// TIA Portal project "立体仓库与堆垛系统_V18" (V18)

(* hardware
DEVICE "S7-1200 station_1"  S7-1200 Station
   slot 0: "Rack_0"  S7-1200 Rack  Rack  V1.0
   slot 1: "PLC_1"  CPU 1214C DC/DC/DC  6ES7 214-1AG31-0XB0  V3.0
DEVICE "HMI_1"  TP700 Comfort
   slot 0: "HMI_1"  TP700 Comfort  6AV2 124-0GC01-0AX0  16.0.0.0
   slot 1: "HMI_RT_1"  TP700 Comfort  6AV2 124-0GC01-0AX0  16.0.0.0
   slot 5: "HMI_1.IE_CP_1"  PROFINET Interface  16.0.0.0
      slot 1: "PROFINET Interface_1"  PROFINET Interface
         slot 1: "Port_1"  Port
         slot 2: "Port_2"  Port
   slot 7: "HMI_1.MPI/DP_CP_1"  MPI/DP Interface  16.0.0.0
DEVICE "GSD device_1"  GSD.Device.PN
   slot 0: "机架"  Rack  V1.0
   slot 0: "gl20-pn"  GL20  INOVANCE GL20-PN
      slot 0: "Standard, 1 port"  Standard, 1 port
      slot 1: "Interface"  Interface
         slot 1: "Port 1"  Port 1
         slot 2: "Port 2"  Port 2
   slot 1: " 1600END_1"  1600END
      slot 0: " 1600END"  1600END
   slot 2: " 1600END_2"  1600END
      slot 0: " 1600END"  1600END
   slot 3: " 0800END_1"  0800END
      slot 0: " 0800END"  0800END
   slot 4: " 0016ETN_1"  0016ETN
      slot 0: " 0016ETN"  0016ETN
DEVICE "GSD device_2"  GSD.Device.PN
   slot 0: "机架"  Rack  V1.0
   slot 0: "GL20-pn2"  GL20  INOVANCE GL20-PN
      slot 0: "Standard, 1 port"  Standard, 1 port
      slot 1: "Interface"  Interface
         slot 1: "Port 1"  Port 1
         slot 2: "Port 2"  Port 2
   slot 1: " 1600END_1"  1600END
      slot 0: " 1600END"  1600END
   slot 2: " 0800END_1"  0800END
      slot 0: " 0800END"  0800END
   slot 3: " 0016ETN_1"  0016ETN
      slot 0: " 0016ETN"  0016ETN
*)

// ===== PLC "PLC_1"  CPU 1214C DC/DC/DC =====

VAR_GLOBAL   // PLC tag table "默认变量表"
   "上升按钮" AT %I4.5 : Bool;
   "下降按钮" AT %I4.4 : Bool;
   "自动手动切换按钮" AT %I5.4 : Bool;
   "进货台正转按钮" AT %I4.0 : Bool;
   "进货链运行按钮" AT %I4.1 : Bool;
   "向后按钮" AT %I4.2 : Bool;
   "向前按钮" AT %I4.3 : Bool;
   "右移按钮" AT %I4.6 : Bool;
   "左移按钮" AT %I4.7 : Bool;
   "进货台反转按钮" AT %I5.0 : Bool;
   "出货链运行按钮" AT %I5.1 : Bool;
   "出货台正转按钮" AT %I5.2 : Bool;
   "出货台反转按钮" AT %I5.3 : Bool;
   "Encoder A pulse" AT %I0.0 : Bool;
   "Encoder B pulse" AT %I0.2 : Bool;
   "Shipment in place detection" AT %I2.2 : Bool;
   "enter table limit position" AT %I2.3 : Bool;
   "enter table Zero position" AT %I2.4 : Bool;
   "Incoming goods in place detection" AT %I2.5 : Bool;
   "Left limit of x-axis" AT %I2.6 : Bool;
   "Lower limit of y-axis" AT %I2.7 : Bool;
   "Platform front and back position judgment" AT %I3.0 : Bool;
   "Platform median detection" AT %I3.1 : Bool;
   "Platform behind Limit Position" AT %I3.2 : Bool;
   "Platform Front Limit Position" AT %I3.3 : Bool;
   "Right limit x-axis" AT %I3.4 : Bool;
   "shipping table  Zero position" AT %I3.5 : Bool;
   "shipping table  limit position" AT %I3.6 : Bool;
   "highlimit y-axis" AT %I3.7 : Bool;
   "急停按钮" AT %I5.5 : Bool;
   "16.space in" AT %I6.0 : Bool;   // 16仓库输入
   "15.space in" AT %I6.1 : Bool;   // 15仓库输入
   "14.space in" AT %I6.2 : Bool;   // 14仓库输入
   "13.space in" AT %I6.3 : Bool;   // 13仓库输入
   "4.space in" AT %I6.4 : Bool;   // 4仓库输入
   "3.space in" AT %I6.5 : Bool;   // 3仓库输入
   "2.space in" AT %I6.6 : Bool;   // 2仓库输入
   "1.space in" AT %I6.7 : Bool;   // 1仓库输入
   "Y-axis stepping pulse" AT %Q0.2 : Bool;
   "Y-axis stepping direction" AT %Q0.3 : Bool;
   "High scan" AT %Q3.4 : Bool;
   "Low scan" AT %Q3.2 : Bool;
   "Mid scan" AT %Q3.3 : Bool;
   "进货台逆时针" AT %Q2.3 : Bool;
   "进货台顺时针" AT %Q2.2 : Bool;
   "进货台电机驱动" AT %Q2.4 : Bool;
   "平台向后运行" AT %Q2.1 : Bool;
   "平台向前运行" AT %Q2.0 : Bool;
   "轴向右运行" AT %Q2.6 : Bool;
   "轴向左运行" AT %Q2.5 : Bool;
   "出货台电机驱动" AT %Q3.1 : Bool;
   "出货台顺时针" AT %Q2.7 : Bool;
   "出货台逆时针" AT %Q3.0 : Bool;
   "步进电机硬件限位辅助" AT %Q3.5 : Bool;
   "Enable manual" AT %M0.4 : Bool;
   "Alarm level" AT %MB100 : Byte;
   "Alarm level 1" AT %M101.0 : Bool;
   "Alarm level 2" AT %M101.1 : Bool;
   "Disconnect Automatic" AT %M101.2 : Bool;
   "Emergency stop system" AT %M101.3 : Bool;
   "组态报警" AT %M101.4 : Bool;
   "触摸屏进入自动" AT %M0.1 : Bool;
   "automatic mode" AT %M0.0 : Bool;
   "manual mode" AT %M0.2 : Bool;
   "stoprightnow" AT %M0.3 : Bool;
   "outover" AT %M0.5 : Bool;
   "inover" AT %M0.6 : Bool;
   "outrequests" AT %M0.7 : Bool;
   "inrequests" AT %M1.0 : Bool;
   "inmod" AT %M1.1 : Bool;
   "outmod" AT %M1.2 : Bool;
   "Warehouse vacancies" AT %M1.3 : Bool;
   "space1" AT %M2.0 : Bool;   // 仓口1
   "space2" AT %M2.1 : Bool;
   "space3" AT %M2.2 : Bool;
   "space4" AT %M2.3 : Bool;
   "space5" AT %M2.4 : Bool;
   "space6" AT %M2.5 : Bool;
   "space7" AT %M2.6 : Bool;
   "space8" AT %M2.7 : Bool;
   "space9" AT %M3.0 : Bool;
   "space10" AT %M3.1 : Bool;
   "space11" AT %M3.2 : Bool;
   "space12" AT %M3.3 : Bool;
   "space13" AT %M3.4 : Bool;
   "space14" AT %M3.5 : Bool;
   "space15" AT %M3.6 : Bool;
   "space16" AT %M3.7 : Bool;
   "space17" AT %M4.0 : Bool;
   "space18" AT %M4.1 : Bool;
   "space19" AT %M4.2 : Bool;
   "space20" AT %M4.3 : Bool;
   "shelf1.NO1" AT %MB2 : USInt;
   "shelf1.NO2" AT %MB3 : USInt;
   "shelf2" AT %MB4 : USInt;
   "移动至货仓8" AT %M10.0 : Bool;
   "移动至货仓7" AT %M10.1 : Bool;
   "移动至货仓6" AT %M10.2 : Bool;
   "移动至货仓5" AT %M10.3 : Bool;
   "移动至货仓4" AT %M10.4 : Bool;
   "移动至货仓3" AT %M10.5 : Bool;
   "移动至货仓2" AT %M10.6 : Bool;
   "移动至货仓1" AT %M10.7 : Bool;
   "移动至货仓16" AT %M11.0 : Bool;
   "移动至货仓15" AT %M11.1 : Bool;
   "移动至货仓14" AT %M11.2 : Bool;
   "移动至货仓13" AT %M11.3 : Bool;
   "移动至货仓12" AT %M11.4 : Bool;
   "移动至货仓11" AT %M11.5 : Bool;
   "移动至货仓10" AT %M11.6 : Bool;
   "移动至货仓9" AT %M11.7 : Bool;
   "移动至货仓17" AT %M12.0 : Bool;
   "移动至货仓18" AT %M12.1 : Bool;
   "移动至货仓19" AT %M12.2 : Bool;
   "移动至货仓20" AT %M12.3 : Bool;
   "backhome" AT %M200.0 : Bool;
   "higher limit of y-axis.sav" AT %M320.2 : Bool;
   "manual_up" AT %M200.3 : Bool;
   "Manual_descent" AT %M200.4 : Bool;
   "Setting Y displacement" AT %MD210 : Real;
   "frontbackO" AT %M13.0 : Bool;
   "behindbackO" AT %M13.1 : Bool;
   "frontlimitgo" AT %M13.2 : Bool;
   "behindlimitgo" AT %M13.3 : Bool;
   "front and back pos judge.sav" AT %M13.4 : Bool;
   "停止回原点前半边" AT %M13.6 : Bool;   // +
   "停止回原点后半轴" AT %M13.7 : Bool;
   "平台前后位判断存(1)" AT %M14.0 : Bool;
   "Pulse A-encoder value" AT %ID1000 : UDInt;
   "Setting X displacement" AT %MD220 : UDInt;
   "insteps.sav" AT %MB5 : USInt;
   "instep1" AT %M15.0 : Bool;
   "instep2" AT %M15.1 : Bool;
   "instep3" AT %M15.2 : Bool;
   "instep4" AT %M15.3 : Bool;
   "instep5" AT %M15.4 : Bool;
   "自动回原点上升" AT %M200.5 : Bool;
   "绝对位移" AT %M200.6 : Bool;
   "回相对原点O" AT %M200.7 : Bool;
   "向O上升" AT %M6.0 : Bool;
   "远O下降" AT %M6.1 : Bool;
   "确认复位" AT %M6.2 : Bool;
   "Tag_1" AT %M17.0 : Bool;
   "调试专用" AT %M9.0 : Bool;
   "Z轴电机初始态完成" AT %M8.1 : Bool;
   "限制使用现场手自动" AT %M1.4 : Bool;
   "AUTO/manual" AT %M1.5 : Bool;
   "in_Pick Pos Completion" AT %M8.0 : Bool;
   "X auto left" AT %M7.0 : Bool;
   "X auto right" AT %M7.1 : Bool;
   "X-axis motion end" AT %M7.2 : Bool;
   "Y-axis motion end" AT %M7.3 : Bool;
   "X-axis right motion lock" AT %M7.4 : Bool;
   "X-axis left motion lock" AT %M7.5 : Bool;
   "instep6" AT %M15.5 : Bool;
   "instep7" AT %M15.6 : Bool;
   "AUTObehindlimitgo" AT %M7.6 : Bool;
   "AUTObehindbackO" AT %M7.7 : Bool;
   "AUTOfrontlimitgo" AT %M14.1 : Bool;
   "AUTOfrontbackO" AT %M14.2 : Bool;
   "停止轴" AT %M8.2 : Bool;
   "instep8" AT %M15.7 : Bool;
   "instep9" AT %M16.0 : Bool;
   "instep10" AT %M16.1 : Bool;
   "步进电机绝对位移ERROR-ID" AT %MD1000 : DWord;
   "Y_coordinate" AT %MD230 : Real;
   "X_coordinate" AT %MD240 : UDInt;
   "Tscan_over" AT %M17.1 : Bool;
   "Tscan_ET" AT %MD1004 : Time;
   "LV.highset" AT %M17.2 : Bool;
   "LV.midset" AT %M17.3 : Bool;
   "LV.lowset" AT %M17.4 : Bool;
   "instep11" AT %M16.2 : Bool;
   "endLOCAT.X" AT %MD250 : UDInt;
   "endLOCAT.Y" AT %MD260 : Real;
   "instep12" AT %M16.3 : Bool;
   "instep13" AT %M16.4 : Bool;
   "instep14" AT %M16.5 : Bool;
   "instep15" AT %M16.6 : Bool;
   "LOWTIME" AT %MD270 : Time;
   "MIDTIME" AT %MD274 : Time;
   "HIGHTIME" AT %MD278 : Time;
   "mov_to1" AT %M110.0 : Bool;   // 人机交互-组态
   "mov_to2" AT %M110.1 : Bool;
   "mov_to3" AT %M110.2 : Bool;
   "mov_to4" AT %M110.3 : Bool;
   "mov_to5" AT %M110.4 : Bool;
   "mov_to6" AT %M110.5 : Bool;
   "mov_to7" AT %M110.6 : Bool;
   "mov_to8" AT %M110.7 : Bool;
   "mov_to9" AT %M111.0 : Bool;
   "mov_to10" AT %M111.1 : Bool;
   "mov_to11" AT %M111.2 : Bool;
   "mov_to12" AT %M111.3 : Bool;
   "mov_to13" AT %M111.4 : Bool;
   "mov_to14" AT %M111.5 : Bool;
   "mov_to15" AT %M111.6 : Bool;
   "mov_to16" AT %M111.7 : Bool;
   "mov_to17" AT %M112.0 : Bool;
   "mov_to18" AT %M112.1 : Bool;
   "mov_to19" AT %M112.2 : Bool;
   "mov_to20" AT %M112.3 : Bool;
   "outgoodsexist" AT %M17.5 : Bool;
   "outsteps.sav" AT %MB18 : USInt;
   "outstep1" AT %M19.0 : Bool;
   "outstep2" AT %M19.1 : Bool;
   "outstep3" AT %M19.2 : Bool;
   "outstep4" AT %M19.3 : Bool;
   "outstep5" AT %M19.4 : Bool;
   "outstep6" AT %M19.5 : Bool;
   "outstep7" AT %M19.6 : Bool;
   "outstep8" AT %M19.7 : Bool;
   "outstep9" AT %M20.0 : Bool;
   "outstep10" AT %M20.1 : Bool;
   "outstep11" AT %M20.2 : Bool;
   "outstep12" AT %M20.3 : Bool;
   "outstep13" AT %M20.4 : Bool;
   "outstep14" AT %M20.5 : Bool;
   "outstep15" AT %M20.6 : Bool;
   "out_Pick Pos Completion" AT %M17.6 : Bool;
   "opt_interrupt" AT %M17.7 : Bool;
   "outstep16" AT %M20.7 : Bool;
   "inset_running" AT %M21.0 : Bool;
   "outget_running" AT %M21.1 : Bool;
   "WillLOCAT.X" AT %MD282 : UDInt;
   "WillLOCAT.Y" AT %MD286 : Real;
   "error_goodslose(out.mod)" AT %M21.2 : Bool;
   "OUTlosttime" AT %MD1008 : Time;
   "error_spacewrong(In.mod)" AT %M21.3 : Bool;
   "warn_NOspace(In.mod)" AT %M21.4 : Bool;
   "coverchoicehmi" AT %M21.5 : Bool;
   "INlosttime" AT %MD1012 : Time;
   "error_goodslose(IN.mod)" AT %M21.6 : Bool;
   "error_spacewrong(out.mod)" AT %M21.7 : Bool;
   "进货台正转HMI" AT %M30.0 : Bool;
   "进货台反转HMI" AT %M30.1 : Bool;
   "出货台正转HMI" AT %M30.2 : Bool;
   "出货台反转HMI" AT %M30.3 : Bool;
   "进货链运行HMI" AT %M30.4 : Bool;
   "出货链运行HMI" AT %M30.5 : Bool;
   "左移HMI" AT %M30.6 : Bool;
   "右移HMI" AT %M30.7 : Bool;
   "上升HMI" AT %M31.0 : Bool;
   "下降HMI" AT %M31.1 : Bool;
   "向前HMI" AT %M31.2 : Bool;
   "向后HMI" AT %M31.3 : Bool;
   "System_Byte" AT %MB500 : Byte;
   "启动标志点" AT %M400.0 : Bool;
   "循环标志位" AT %M400.1 : Bool;
   "停止" AT %M400.2 : Bool;
   "复位完成" AT %M400.5 : Bool;
   "Tag_2" AT %M400.4 : Bool;
   "Tag_3" AT %M400.6 : Bool;
   "System_Byte(1)" AT %MB1 : Byte;
   "FirstScan" AT %M500.0 : Bool;
   "DiagStatusUpdate" AT %M500.1 : Bool;
   "AlwaysTRUE" AT %M500.2 : Bool;
   "AlwaysFALSE" AT %M500.3 : Bool;
END_VAR

VAR_GLOBAL   // PLC tag table "gl20-np2输出"
   "进" AT %Q4.0 : Bool;
   "推" AT %Q4.1 : Bool;
   "变频器（黄）" AT %Q4.2 : Bool;
   "链运行" AT %Q4.3 : Bool;
   "码垛升" AT %Q4.4 : Bool;
   "挡板挡" AT %Q4.5 : Bool;
   "平台升" AT %Q4.6 : Bool;
   "放" AT %Q4.7 : Bool;
   "退" AT %Q5.0 : Bool;
   "回" AT %Q5.1 : Bool;
   "变频器（橙）" AT %Q5.2 : Bool;
   "带运行" AT %Q5.3 : Bool;
   "码垛降" AT %Q5.4 : Bool;
   "挡板回" AT %Q5.5 : Bool;
   "平台降" AT %Q5.6 : Bool;
   "货转向" AT %Q5.7 : Bool;
END_VAR

VAR_GLOBAL   // PLC tag table "gl20-np2输入"
   "(n)" AT %I7.0 : Bool;
   "码垛升到位传感器(h)" AT %I7.1 : Bool;
   "码垛到位传感器(b)" AT %I7.2 : Bool;
   "推中到位传感器(d)" AT %I7.3 : Bool;
   "推到位传感器(j)" AT %I7.4 : Bool;
   "码垛下降到位传感器(i)" AT %I7.5 : Bool;
   "平台检测光电传感器(L)" AT %I7.6 : Bool;
   "平台上到位传感器(0)" AT %I7.7 : Bool;
   "挡板挡到位(m)" AT %I8.0 : Bool;
   "码垛输入传感器(a)" AT %I8.1 : Bool;
   "回到位传感器(c)" AT %I8.2 : Bool;
   "推到位传感器(e)" AT %I8.3 : Bool;
   "退到位传感器(f)" AT %I8.4 : Bool;
   "码垛高度匹配传感器(g)" AT %I8.5 : Bool;
   "平台到位传感器(k)" AT %I8.6 : Bool;
   "平台下到位传感器(p)" AT %I8.7 : Bool;
   "手动自动" AT %I9.0 : Bool;
END_VAR

DATA_BLOCK "Locat"   // DB11
{ S7_Optimized_Access := 'TRUE' }
VERSION : 0.1
   VAR RETAIN
      "shelf  X axis" : Array[0..19] of UDInt;
      "shelf  Y axis" : Array[0..19] of Real;
   END_VAR
BEGIN
   "shelf  X axis"[0] := 1362;
   "shelf  X axis"[1] := 1362;
   "shelf  X axis"[2] := 1061;
   "shelf  X axis"[3] := 1061;
   "shelf  X axis"[4] := 929;
   "shelf  X axis"[5] := 929;
   "shelf  X axis"[6] := 929;
   "shelf  X axis"[7] := 764;
   "shelf  X axis"[8] := 764;
   "shelf  X axis"[9] := 633;
   "shelf  X axis"[10] := 633;
   "shelf  X axis"[11] := 633;
   "shelf  X axis"[12] := 466;
   "shelf  X axis"[13] := 466;
   "shelf  X axis"[14] := 334;
   "shelf  X axis"[15] := 334;
   "shelf  X axis"[16] := 334;
   "shelf  X axis"[17] := 34;
   "shelf  X axis"[18] := 34;
   "shelf  X axis"[19] := 34;
   "shelf  Y axis"[0] := -263.0;
   "shelf  Y axis"[1] := -130.0;
   "shelf  Y axis"[6] := 2.5;
   "shelf  Y axis"[5] := -130.0;
   "shelf  Y axis"[4] := -263.0;
   "shelf  Y axis"[3] := -130.0;
   "shelf  Y axis"[2] := -263.0;
   "shelf  Y axis"[7] := -263.0;
   "shelf  Y axis"[8] := -130.0;
   "shelf  Y axis"[9] := -263.0;
   "shelf  Y axis"[10] := -130.0;
   "shelf  Y axis"[11] := 2.5;
   "shelf  Y axis"[12] := -263.0;
   "shelf  Y axis"[13] := -130.0;
   "shelf  Y axis"[14] := -263.0;
   "shelf  Y axis"[15] := -130.0;
   "shelf  Y axis"[16] := 2.5;
   "shelf  Y axis"[17] := -263.0;
   "shelf  Y axis"[18] := -130.0;
   "shelf  Y axis"[19] := 2.5;
END_DATA_BLOCK

DATA_BLOCK "mov choice"   // DB12
{ S7_Optimized_Access := 'TRUE' }
VERSION : 0.1
   VAR RETAIN
      NO : Array[0..19] of Bool;
   END_VAR
   VAR
      i : USInt;
      WZ : USInt;
   END_VAR
BEGIN
END_DATA_BLOCK

// folder: System blocks/Program resources

DATA_BLOCK "复位协助z轴"   // DB7
{ S7_Optimized_Access := 'TRUE' }
AUTHOR : Simatic
FAMILY : IEC
NAME : IEC_TMR
VERSION : 1.0
// stored: InstanceOfName IEC_TIMER
"IEC_TIMER"
BEGIN
END_DATA_BLOCK

DATA_BLOCK "脉冲定时底"   // DB8
{ S7_Optimized_Access := 'TRUE' }
AUTHOR : Simatic
FAMILY : IEC
NAME : IEC_TMR
VERSION : 1.0
// stored: InstanceOfName IEC_TIMER
"IEC_TIMER"
BEGIN
END_DATA_BLOCK

DATA_BLOCK "脉冲定时中"   // DB9
{ S7_Optimized_Access := 'TRUE' }
AUTHOR : Simatic
FAMILY : IEC
NAME : IEC_TMR
VERSION : 1.0
// stored: InstanceOfName IEC_TIMER
"IEC_TIMER"
BEGIN
END_DATA_BLOCK

DATA_BLOCK "脉冲定时高"   // DB10
{ S7_Optimized_Access := 'TRUE' }
AUTHOR : Simatic
FAMILY : IEC
NAME : IEC_TMR
VERSION : 1.0
// stored: InstanceOfName IEC_TIMER
"IEC_TIMER"
BEGIN
END_DATA_BLOCK

DATA_BLOCK "time_scan_houseware"   // DB13
{ S7_Optimized_Access := 'TRUE' }
AUTHOR : Simatic
FAMILY : IEC
NAME : IEC_TMR
VERSION : 1.0
// stored: InstanceOfName IEC_TIMER
"IEC_TIMER"
BEGIN
END_DATA_BLOCK

DATA_BLOCK "NOgoodsTON"   // DB15
{ S7_Optimized_Access := 'TRUE' }
AUTHOR : Simatic
FAMILY : IEC
NAME : IEC_TMR
VERSION : 1.0
// stored: InstanceOfName IEC_TIMER
"IEC_TIMER"
BEGIN
END_DATA_BLOCK

// folder: 堆垛系统

DATA_BLOCK "数据块"   // DB16
{ S7_Optimized_Access := 'TRUE' }
VERSION : 0.1
   VAR
      标志位 : Array[1..30] of Bool;
      沿 : Array[1..9] of Bool;
      定时器 : Array[1..6] of IEC_TIMER;
      码垛数量 : Int;
      当前时间 : Time;
      限制 : Bool;
      码垛总数量 : Int;
      余数 : Int;
   END_VAR
BEGIN
END_DATA_BLOCK

DATA_BLOCK "输出数据块"   // DB17
{ S7_Optimized_Access := 'FALSE' }
VERSION : 0.1
   VAR
      带运行 : Bool;
      推 : Bool;
      回1 : Bool;
      回2 : Bool;
      平台降 : Bool;
      平台升1 : Bool;
      平台升2 : Bool;
      放 : Bool;
      链运行 : Bool;
      链运行2 : Bool;
      码垛降 : Bool;
      码垛升1 : Bool;
      码垛升2 : Bool;
      码垛进 : Bool;
      码垛退1 : Bool;
      码垛退2 : Bool;
      挡板挡 : Bool;
      挡板回1 : Bool;
      挡板回2 : Bool;
   END_VAR
BEGIN
END_DATA_BLOCK

// folder: (top level)

DATA_BLOCK "轴_1"   // DB1, Motion_DB
{ S7_Optimized_Access := 'TRUE' }
AUTHOR : SIMATIC
FAMILY : BasicMC
NAME : TO_PTO
VERSION : 3.0
// stored: InstanceOfName TO_Axis_PTO
"TO_Axis_PTO"
BEGIN
   // Axis.OnlinePtoIndexCU = 1
   // Axis.DirectionHwcnAddressCU = Q0.3
   // Axis.PulseHwcnAddressCU = Q0.2
   // Pulse.MinDeltaDeltaFrequencyCU = 0.004
   // Pulse.MaxDeltaDeltaFrequencyCU = 1.0E+10
   // Pulse.MinDeltaFrequencyCU = 0.005
   // Pulse.MaxDeltaFrequencyCU = 9.5E+9
   // Pulse.MinFrequencyCU = 1.0
   // Pulse.MaxFrequencyCU = 100000.0
   // Pulse.OutputSourceCU = 16#0000_0000
   // Axis.SelectPTO = 1
END_DATA_BLOCK

FUNCTION "Auto Out_ware Main Program" : Void   // FC1, SCL
{ S7_Optimized_Access := 'TRUE' }
VERSION : 0.1
BEGIN
   "Shelf Path Selection Subroutine"();//必须进入出库模式才可以访问本页面
   // "opt_interrupt"=1时进入选择，面板变量会,仅在完成正在执行的出库工作或首次使用出库模式后可激活，更新预定的出库序列
   // 不要同时按"movtoxxxx"和"opt_interrupt:=0".此操作不规范，系统会对此进行紧急停止处理。
   IF "outrequests" = 1 AND "outover" = 1 AND "outsteps.sav" = 0 AND "outgoodsexist"AND "opt_interrupt"=0 THEN
       "outsteps.sav" := 1;
       "outover" := 0;
       "coverchoicehmi" := 0;// 关闭选择面板
   END_IF;
   IF "opt_interrupt"=1 AND "outover" = 1 THEN
       "coverchoicehmi" := 1; // 组态里打开选择面板，才可以选择或取消接下来的取货位置
       ;
   END_IF;


   CASE "outsteps.sav" OF
           //取货步
       1:"outstep1" := 1;
           "out_Pick Pos Completion" := "X-axis motion end" AND "Y-axis motion end";
       2:"outstep2" := 1;
       3:"outstep3" := 1;
       4:"outstep4" := 1;
       5:"outstep5" := 1;
       6:"outstep6" := 1;
       7:"outstep7" := 1;
       8:"outstep8" := 1;
       9:"outstep9" := 1;
       10:"outstep10" := 1;
           "out_Pick Pos Completion" := "X-axis motion end" AND "Y-axis motion end";
       11:"outstep11" := 1;
       12:"outstep12" := 1;
       13:"outstep13" := 1;
       14:"outstep14" := 1;
       15:
           "outstep15" := 1;
       16:
           "outstep16" := 1;
       17:
           "outsteps.sav" := 0; // 步序复位
           "outover" := 1;
           IF "outgoodsexist"=0 THEN
               "mov_to13" := 0;
               "mov_to17" := 0;
               "mov_to14" := 0;
               "mov_to18" := 0;
               "mov_to1" := 0;
               "mov_to5" := 0;
               "mov_to9" := 0;
               "mov_to15" := 0;
               "mov_to19" := 0;
               "mov_to2" := 0;
               "mov_to6" := 0;
               "mov_to10" := 0;
               "mov_to16" := 0;
               "mov_to20" := 0;
               "mov_to3" := 0;
               "mov_to7" := 0;
               "mov_to11" := 0;
               "mov_to4" := 0;
               "mov_to8" := 0;
               "mov_to12" := 0;
               // Statement section IF
               ;
           END_IF;
       ELSE
           "outsteps.sav" := 0; // 步序复位
           "outover" := 1;

   END_CASE;

   //出库步序1取货开始
   IF "outstep1" AND ("out_Pick Pos Completion" = 0) THEN
       "Z-axis motor subroutine"();
       IF  "outget_running"=0 OR ("WillLOCAT.X" = "X_coordinate"AND "WillLOCAT.Y" = "Y_coordinate") THEN
           IF "endLOCAT.X" = "X_coordinate" THEN
               // 不需要左右移动直接取
               "Setting Y displacement" := ("Y_coordinate" - 15.0);
               "Y-axis stepper motor subroutine"();
               "X-axis motion end" := 1;
               "WillLOCAT.X" := "X_coordinate";
               "WillLOCAT.Y" := "Y_coordinate";
               "outget_running" := 1;
           ELSE
               //mov后取        
               "Setting X displacement" := "X_coordinate";
               "Setting Y displacement" := ("Y_coordinate" - 15.0);
               "X-axis motor encoder group subroutine"();
               "Y-axis stepper motor subroutine"();
               "WillLOCAT.X" := "X_coordinate";
               "WillLOCAT.Y" := "Y_coordinate";
               "outget_running" := 1;
           END_IF;
       ELSE
           "stoprightnow" := 1;
           "error_spacewrong(out.mod)" := 1;

       END_IF;



   ELSIF "outstep1" AND ("out_Pick Pos Completion" = 1) THEN
       "outstep1" := 0;
       "outsteps.sav" := "outsteps.sav" + 1;
       "Setting Y displacement" := -120;
       "Y-axis stepper motor subroutine"();
       "X-axis motion end" := 0;
       "X-axis left motion lock" := 0;
       "X-axis right motion lock" := 0;
       "Setting X displacement" := 0;
       "endLOCAT.X" :="X_coordinate";
       "endLOCAT.Y" := "Y_coordinate";
       "outget_running" := 0;
   END_IF;
   //出库步序2选择货架
   IF "outstep2" THEN
       IF    "WillLOCAT.X" = "X_coordinate"AND "WillLOCAT.Y" = "Y_coordinate"  THEN
           IF "X_coordinate" = 929 OR "X_coordinate" = 633 OR "X_coordinate" = 334 OR "X_coordinate" = 34 THEN
               "outstep2" := 0;
               "outsteps.sav" := "outsteps.sav" + 4;
           ELSIF "X_coordinate" = 1362 OR "X_coordinate" = 1061 OR "X_coordinate" = 764 OR "X_coordinate" = 466 THEN
               "outstep2" := 0;
               "outsteps.sav" := "outsteps.sav" + 1;
               ;
           END_IF;  // Statement section IF
       ELSE
           "stoprightnow" := 1;
           "error_spacewrong(out.mod)" := 1;
       END_IF;



   END_IF;
       //取货架2
       //出库步序3
       IF "outstep3" AND ("Platform Front Limit Position" = 0) THEN
           "AUTOfrontlimitgo" := 1;
           "Z-axis motor subroutine"();
       ELSIF "outstep3" AND ("Platform Front Limit Position" = 1) THEN
           "AUTOfrontlimitgo" := 0;
           "outstep3" := 0;
           "outsteps.sav" := "outsteps.sav" + 1;
       END_IF;
       //出库步序4
       IF "outstep4" AND ("Y-axis motion end" = 0) THEN
           "Z-axis motor subroutine"();
               "Setting Y displacement" := "Y_coordinate";
               "Y-axis stepper motor subroutine"();
       ELSIF "outstep4" AND ("Y-axis motion end" = 1) THEN
           "outstep4" := 0;
           "outsteps.sav" := "outsteps.sav" + 1;
           "Setting Y displacement" := -120;
           "Y-axis stepper motor subroutine"();
       END_IF;
       //出库步序5
       IF "outstep5" AND ("Platform Front Limit Position" = 1 OR "frontbackO" = 1) THEN
           "AUTOfrontbackO" := 1;
           "Z-axis motor subroutine"();
       ELSIF "outstep5" AND ("Platform Front Limit Position" = 0 AND "frontbackO" = 0) THEN
           "AUTOfrontbackO" := 0;
           "outstep5" := 0;
           "outsteps.sav" := "outsteps.sav" + 4;
       END_IF;
       //取货架1
       //出库步序6
       IF "outstep6" AND ("Platform behind Limit Position" = 0) THEN
           "AUTObehindlimitgo" := 1;
           "Z-axis motor subroutine"();
       ELSIF "outstep6" AND ("Platform behind Limit Position" = 1) THEN
           "AUTObehindlimitgo" := 0;
           "outstep6" := 0;
           "outsteps.sav" := "outsteps.sav" + 1;
       END_IF;
       //出库步序7
       IF "outstep7" AND ("Y-axis motion end" = 0) THEN
           "Z-axis motor subroutine"();
               "Setting Y displacement" := "Y_coordinate";
               "Y-axis stepper motor subroutine"();
       ELSIF "outstep7" AND ("Y-axis motion end" = 1) THEN
           "outstep7" := 0;
           "outsteps.sav" := "outsteps.sav" + 1;
           "Setting Y displacement" := -120;
           "Y-axis stepper motor subroutine"();
       END_IF;
       //出库步序8
       IF "outstep8" AND ("Platform behind Limit Position" = 1 OR "behindbackO" = 1) THEN
           "AUTObehindbackO" := 1;
           "Z-axis motor subroutine"();
       ELSIF "outstep8" AND ("Platform behind Limit Position" = 0 AND "behindbackO" = 0) THEN
           "AUTObehindbackO" := 0;
           "outstep8" := 0;
           "outsteps.sav" := "outsteps.sav" + 1;
       END_IF;
       //出库步序9
       IF "outstep9" AND ("shipping table  Zero position" = 0) THEN
           "出货台逆时针" := 1 AND ("stoprightnow" = 0);
       ELSIF "outstep9" AND ("shipping table  Zero position" = 1) THEN
           "出货台逆时针" := 0;
           "outstep9" := 0;
           "outsteps.sav" := "outsteps.sav" + 1;
       END_IF;
       //出库步序10
       IF "outstep10" AND ("out_Pick Pos Completion" = 0) THEN
           "Z-axis motor subroutine"();
           IF "endLOCAT.X" <= 40 AND "endLOCAT.Y" = 2.5 THEN
               "Setting Y displacement" := -260;
               "Y-axis stepper motor subroutine"();
               "X-axis motion end" := 1;
           ELSIF "endLOCAT.X" <= 40 AND "endLOCAT.Y" = -130.0 THEN
               "Setting Y displacement" := -260;
               "Y-axis stepper motor subroutine"();
               "X-axis motion end" := 1;
           ELSIF "endLOCAT.X" <= 40 AND "endLOCAT.Y" = -263.0 THEN
               "Setting Y displacement" := -263;
               "Y-axis stepper motor subroutine"();
               "X-axis motion end" := 1;
           ELSE
               "Setting X displacement" := 35;
               "Setting Y displacement" := -260;
               "X-axis motor encoder group subroutine"();
               "Y-axis stepper motor subroutine"();

           END_IF;
       ELSIF "outstep10" AND ("out_Pick Pos Completion" = 1) THEN
           "outstep10" := 0;
           "outsteps.sav" := "outsteps.sav" + 1;
           "Setting Y displacement" := -120;
           "Y-axis stepper motor subroutine"();
           "X-axis motion end" := 0;
           "X-axis left motion lock" := 0;
           "X-axis right motion lock" := 0;
           "Setting X displacement" := 0;
       END_IF;
       //出库步序11
       IF "outstep11" AND ("Platform Front Limit Position" = 0) THEN
           "AUTOfrontlimitgo" := 1;
           "Z-axis motor subroutine"();
       ELSIF "outstep11" AND ("Platform Front Limit Position" = 1) THEN
           "AUTOfrontlimitgo" := 0;
           "outstep11" := 0;
           "outsteps.sav" := "outsteps.sav" + 1;
       END_IF;
       //出库步序12
       IF "outstep12" AND ("Y-axis motion end" = 0) THEN
           "Z-axis motor subroutine"();
           "Setting Y displacement" := -278;
           "Y-axis stepper motor subroutine"();
       ELSIF "outstep12" AND ("Y-axis motion end" = 1) THEN
           "outstep12" := 0;
           "outsteps.sav" := "outsteps.sav" + 1;
           "Setting Y displacement" := -120;
           "Y-axis stepper motor subroutine"();
       END_IF;
       //出库步序13
       IF "outstep13" AND ("Platform Front Limit Position" = 1 OR "frontbackO" = 1) THEN
           "AUTOfrontbackO" := 1;
           "Z-axis motor subroutine"();
       ELSIF "outstep13" AND ("Platform Front Limit Position" = 0 AND "frontbackO" = 0) THEN
           "AUTOfrontbackO" := 0;
           "outstep13" := 0;
           "outsteps.sav" := "outsteps.sav" + 1;
       END_IF;
       //出库步序14
       IF "outstep14" AND ("Y-axis motion end" = 0) THEN
           "Z-axis motor subroutine"();
           "Setting Y displacement" := -145;
           "Y-axis stepper motor subroutine"();
       ELSIF "outstep14" AND ("Y-axis motion end") THEN
           "outstep14" := 0;
           "outsteps.sav" := "outsteps.sav" + 1;
           "Setting Y displacement" := -120;
           "Y-axis stepper motor subroutine"();
           "endLOCAT.X" := 34;
           "endLOCAT.Y" := -145;
           "WillLOCAT.X" := 0;
           "WillLOCAT.Y" :=0;
       END_IF;
       //出库步序15
       IF "outstep15" AND ("shipping table  limit position" = 0) THEN
           "出货台顺时针" := 1 AND ("stoprightnow" = 0);
       ELSIF "outstep15" AND ("shipping table  limit position" = 1) THEN
           "出货台顺时针" := 0;
           "outstep15" := 0;
           "outsteps.sav" := "outsteps.sav" + 1;
       END_IF;
       //出库步序16
       "NOgoodsTON".TON(IN := ("outstep16" AND NOT "Shipment in place detection"),
                        PT := T#30s,
                        Q => "error_goodslose(out.mod)",
                        ET => "OUTlosttime");
       IF "outstep16" AND ("Shipment in place detection" = 0) THEN
           "出货台电机驱动" := 1 AND ("stoprightnow" = 0);
           "stoprightnow" := "error_goodslose(out.mod)";
       ELSIF "outstep16" AND ("Shipment in place detection" = 1) THEN
           "出货台电机驱动" := 0;
           "outstep16" := 0;
           "outsteps.sav" := "outsteps.sav" + 1;
       END_IF;
END_FUNCTION

FUNCTION "manual control" : Void   // FC2, LAD
{ S7_Optimized_Access := 'TRUE' }
VERSION : 0.1
BEGIN

REGION Network 1 (SCL)
   //手动切换为自动后必须立即进行复位，禁止不复位而立即请求
   IF "自动手动切换按钮" = 0 THEN
       "outmod" := 0;
       "inmod" := 0;
       "inrequests" := 0;
       "outrequests" := 0;
   END_IF;
END_REGION

REGION Network 2
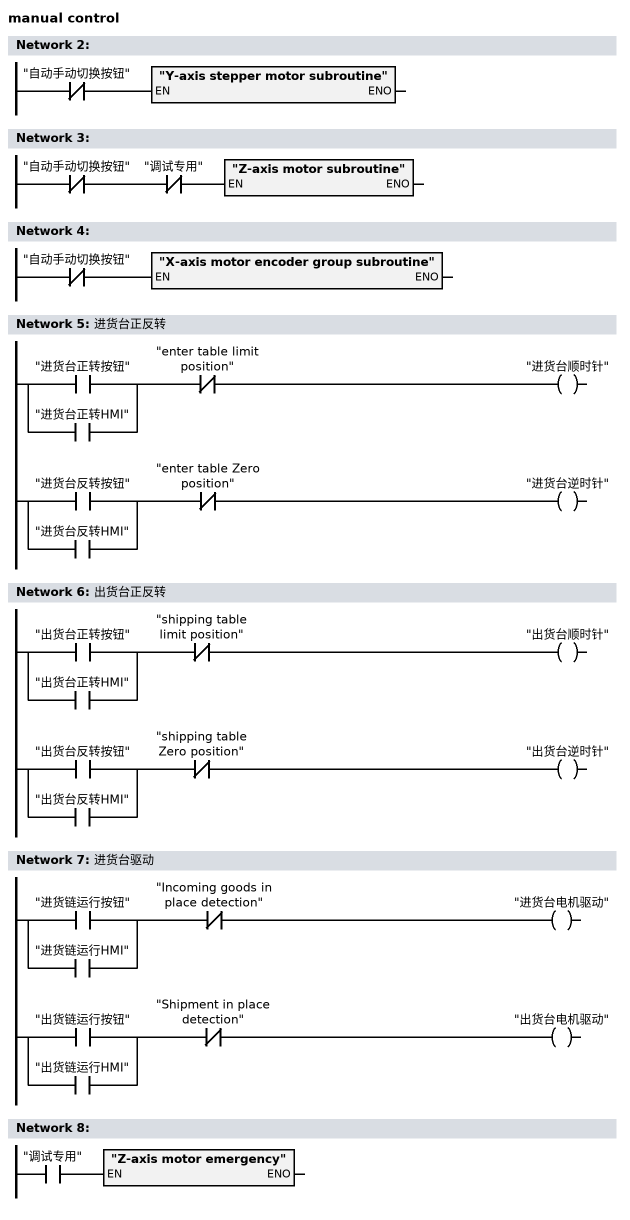
   RUNG wire#powerrail
      I_Contact( "自动手动切换按钮" )
      "Y-axis stepper motor subroutine"()
   END_RUNG
   // the same network as SCL:
   IF NOT "自动手动切换按钮" THEN "Y-axis stepper motor subroutine"(); END_IF;
END_REGION

REGION Network 3
   RUNG wire#powerrail
      I_Contact( "自动手动切换按钮" )
      I_Contact( "调试专用" )
      "Z-axis motor subroutine"()
   END_RUNG
   // the same network as SCL:
   IF NOT "自动手动切换按钮" AND NOT "调试专用" THEN "Z-axis motor subroutine"(); END_IF;
END_REGION

REGION Network 4
   RUNG wire#powerrail
      I_Contact( "自动手动切换按钮" )
      "X-axis motor encoder group subroutine"()
   END_RUNG
   // the same network as SCL:
   IF NOT "自动手动切换按钮" THEN "X-axis motor encoder group subroutine"(); END_IF;
END_REGION

REGION Network 5: 进货台正反转
   RUNG wire#powerrail
      Contact( "进货台正转按钮" )
      wire#w1
      I_Contact( "enter table limit position" )
      Coil( "进货台顺时针" )
   END_RUNG
   RUNG wire#powerrail
      Contact( "进货台正转HMI" )
   END_RUNG wire#w1
   RUNG wire#powerrail
      Contact( "进货台反转按钮" )
      wire#w2
      I_Contact( "enter table Zero position" )
      Coil( "进货台逆时针" )
   END_RUNG
   RUNG wire#powerrail
      Contact( "进货台反转HMI" )
   END_RUNG wire#w2
   // the same network as SCL:
   "进货台顺时针" := ("进货台正转按钮" OR "进货台正转HMI") AND NOT "enter table limit position";
   "进货台逆时针" := ("进货台反转按钮" OR "进货台反转HMI") AND NOT "enter table Zero position";
END_REGION

REGION Network 6: 出货台正反转
   RUNG wire#powerrail
      Contact( "出货台正转按钮" )
      wire#w1
      I_Contact( "shipping table  limit position" )
      Coil( "出货台顺时针" )
   END_RUNG
   RUNG wire#powerrail
      Contact( "出货台正转HMI" )
   END_RUNG wire#w1
   RUNG wire#powerrail
      Contact( "出货台反转按钮" )
      wire#w2
      I_Contact( "shipping table  Zero position" )
      Coil( "出货台逆时针" )
   END_RUNG
   RUNG wire#powerrail
      Contact( "出货台反转HMI" )
   END_RUNG wire#w2
   // the same network as SCL:
   "出货台顺时针" := ("出货台正转按钮" OR "出货台正转HMI") AND NOT "shipping table  limit position";
   "出货台逆时针" := ("出货台反转按钮" OR "出货台反转HMI") AND NOT "shipping table  Zero position";
END_REGION

REGION Network 7: 进货台驱动
   RUNG wire#powerrail
      Contact( "进货链运行按钮" )
      wire#w1
      I_Contact( "Incoming goods in place detection" )
      Coil( "进货台电机驱动" )
   END_RUNG
   RUNG wire#powerrail
      Contact( "进货链运行HMI" )
   END_RUNG wire#w1
   RUNG wire#powerrail
      Contact( "出货链运行按钮" )
      wire#w2
      I_Contact( "Shipment in place detection" )
      Coil( "出货台电机驱动" )
   END_RUNG
   RUNG wire#powerrail
      Contact( "出货链运行HMI" )
   END_RUNG wire#w2
   // the same network as SCL:
   "进货台电机驱动" := ("进货链运行按钮" OR "进货链运行HMI") AND NOT "Incoming goods in place detection";
   "出货台电机驱动" := ("出货链运行按钮" OR "出货链运行HMI") AND NOT "Shipment in place detection";
END_REGION

REGION Network 8
   RUNG wire#powerrail
      Contact( "调试专用" )
      "Z-axis motor emergency"()
   END_RUNG
   // the same network as SCL:
   IF "调试专用" THEN "Z-axis motor emergency"(); END_IF;
END_REGION
END_FUNCTION

FUNCTION "Z-axis motor emergency" : Void   // FC3, LAD
{ S7_Optimized_Access := 'TRUE' }
VERSION : 0.1
   VAR_TEMP   // added for the SCL form of the ladder/FBD networks
      _w1 : Bool;
   END_VAR
BEGIN

REGION Network 1 (SCL)
   "frontbackO" := 0;
   "behindbackO" := 0;
   "frontlimitgo" := 0;
   "behindlimitgo" := 0;
END_REGION

REGION Network 2
   // //当z轴电机出现紧急情况时，先停止再按下调试专用按钮再切手动即可进行微步调试
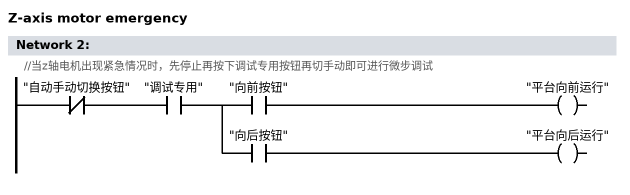
   RUNG wire#powerrail
      I_Contact( "自动手动切换按钮" )
      Contact( "调试专用" )
      wire#w1
      Contact( "向前按钮" )
      Coil( "平台向前运行" )
   END_RUNG
   RUNG wire#w1
      Contact( "向后按钮" )
      Coil( "平台向后运行" )
   END_RUNG
   // the same network as SCL:
   #_w1 := NOT "自动手动切换按钮" AND "调试专用";
   "平台向前运行" := #_w1 AND "向前按钮";
   "平台向后运行" := #_w1 AND "向后按钮";
END_REGION
END_FUNCTION

FUNCTION "system reset" : Void   // FC5, LAD
{ S7_Optimized_Access := 'TRUE' }
VERSION : 0.1
// 紧急情况按停止再复位，如果是z轴紧急则用紧急调试块
BEGIN

REGION Network 1 (SCL): 模式参数初始化
   // 停止情况下仍可按复位进行动作
   "inover" := 1;
   "outover" := 1;
   "outmod" := 0;//清除模式
   "inmod" := 0;
   "inrequests" := 0;//清除请求
   "outrequests" := 0;
   "endLOCAT.X" :=0;
   "endLOCAT.Y" :=0;
   "WillLOCAT.X" := 0;
   "WillLOCAT.Y" := 0;
   "AUTObehindlimitgo" := 0;
   "AUTObehindbackO" := 0;
   "AUTOfrontlimitgo" := 0;
   "AUTOfrontbackO" := 0;
   "Z-axis motor subroutine"();
END_REGION

REGION Network 2 (SCL): 停止手动
   "进货台逆时针" :=0;
   "进货台顺时针" := 0;
   "进货台电机驱动" := 0;
   "出货台顺时针" := 0;
   "出货台逆时针" := 0;
   "出货台电机驱动" := 0;
   "manual_up" := 0;
   "Manual_descent" := 0;
   "error_goodslose(out.mod)":=0;
   "error_spacewrong(out.mod)":=0;
   "error_spacewrong(In.mod)" := 0;
   "error_goodslose(IN.mod)" := 0;
   "warn_NOspace(In.mod)" := 0;
END_REGION

REGION Network 3 (SCL): 自动入库数据复位
   IF "确认复位" THEN
       "insteps.sav" := 0;
       "instep1" := 0;
       "instep2" := 0;
       "instep3" := 0;
       "instep4" := 0;
       "instep5" := 0;
       "instep6" := 0;
       "instep7" := 0;
       "instep8" := 0;
       "instep9" := 0;
       "instep10" := 0;
       "instep11" := 0;
       "instep12" := 0;
       "instep13" := 0;
       "instep14" := 0;
       "instep15" := 0;
       "X auto left" := 0;
       "X auto right" := 0;
       "mov choice".WZ := 0;
       "Warehouse vacancies" := 1;
       //步序三部分复位   
       "X-axis motion end" := 0;
       "X-axis left motion lock" := 0;
       "X-axis right motion lock" := 0;
       "Setting X displacement" := 0;
       // Statement section IF
       "in_Pick Pos Completion" := 0;
       "inset_running" := 0;
   END_IF;
END_REGION

REGION Network 4 (SCL): 自动出库数据复位
   IF "确认复位" THEN
       "outsteps.sav" := 0;
       "outstep1" := 0;
       "outstep2" := 0;
       "outstep3" := 0;
       "outstep4" := 0;
       "outstep5" := 0;
       "outstep6" := 0;
       "outstep7" := 0;
       "outstep8" := 0;
       "outstep9" := 0;
       "outstep10" := 0;
       "outstep11" := 0;
       "outstep12" := 0;
       "outstep13" := 0;
       "outstep14" := 0;
       "outstep15" := 0;
       "outstep16" := 0;
       "X auto left" := 0;
       "X auto right" := 0;
       //部分复位   
       "X-axis motion end" := 0;
       "X-axis left motion lock" := 0;
       "X-axis right motion lock" := 0;
       "Setting X displacement" := 0;
       "outgoodsexist" := 1;
       // Statement section IF
       "out_Pick Pos Completion" := 0;
       "opt_interrupt" := 0;
       "outget_running" := 0;
       //复位出库选择
    "mov_to13":=0;
    "mov_to17" := 0;
    "mov_to14" := 0;
    "mov_to18" := 0;
    "mov_to1" := 0;
    "mov_to5" := 0;
    "mov_to9" := 0;
    "mov_to15" := 0;
    "mov_to19" := 0;
    "mov_to2" := 0;
    "mov_to6" := 0;
    "mov_to10" := 0;
    "mov_to16" := 0;
    "mov_to20" := 0;
    "mov_to3" := 0;
    "mov_to7" := 0;
    "mov_to11" := 0;
    "mov_to4" := 0;
    "mov_to8" := 0;
    "mov_to12" := 0;
   END_IF;
END_REGION

REGION Network 5 (SCL): 复位
   "回相对原点O" := "确认复位"AND"Z轴电机初始态完成" ;
   "Setting Y displacement" := -120;
   "Y-axis stepper motor subroutine"();
   "回相对原点O" := 0;
   "进货台逆时针" := (NOT "enter table Zero position")AND "确认复位"AND"Z轴电机初始态完成" AND "highlimit y-axis"AND "Right limit x-axis";
   "出货台顺时针" := (NOT "shipping table  limit position") AND "确认复位"AND"Z轴电机初始态完成" AND "highlimit y-axis"AND "Right limit x-axis" ;
   "X-axis motor encoder group subroutine"();
END_REGION
END_FUNCTION

FUNCTION "in_out_manage subroutine" : Void   // FC6, SCL
{ S7_Optimized_Access := 'TRUE' }
VERSION : 0.1
BEGIN
   //切换模式前，需要当前模式结束动作才允许切换；中途切换建议复位后再操作。
   IF "inrequests" = 1  AND "outrequests" = 0  AND "stoprightnow"=0 AND "outover" THEN
       "inmod" := 1;
       "outmod" := 0;
       //一旦进入入库模式清空出库选择
       "mov_to13" := 0;
       "mov_to17" := 0;
       "mov_to14" := 0;
       "mov_to18" := 0;
       "mov_to1" := 0;
       "mov_to5" := 0;
       "mov_to9" := 0;
       "mov_to15" := 0;
       "mov_to19" := 0;
       "mov_to2" := 0;
       "mov_to6" := 0;
       "mov_to10" := 0;
       "mov_to16" := 0;
       "mov_to20" := 0;
       "mov_to3" := 0;
       "mov_to7" := 0;
       "mov_to11" := 0;
       "mov_to4" := 0;
       "mov_to8" := 0;
       "mov_to12" := 0;
   END_IF;     
   //出库请求优先级最高，可以在入库模式下直接切换但必须是入库结束后才行。
   IF "outrequests"=1AND "stoprightnow"=0 AND "inover"  THEN
       "outmod" := 1;
       "inmod" := 0;
   END_IF;
END_FUNCTION

FUNCTION "Shelf Path Selection Subroutine" : Void   // FC7, LAD
{ S7_Optimized_Access := 'TRUE' }
VERSION : 0.1
BEGIN

REGION Network 1 (SCL): 入库路径选择自动方案
   IF "inmod" THEN
       "mov choice".NO[0] := NOT "space13";
       "mov choice".NO[1] := NOT "space17";
       "mov choice".NO[2] := NOT "space14";
       "mov choice".NO[3] := NOT "space18";
       "mov choice".NO[4] := NOT "space1";
       "mov choice".NO[5] := NOT "space5";
       "mov choice".NO[6] := NOT "space9";
       "mov choice".NO[7] := NOT "space15";
       "mov choice".NO[8] := NOT "space19";
       "mov choice".NO[9] := NOT "space2";
       "mov choice".NO[10] := NOT "space6";
       "mov choice".NO[11] := NOT "space10";
       "mov choice".NO[12] := NOT "space16";
       "mov choice".NO[13] := NOT "space20";
       "mov choice".NO[14] := NOT "space3";
       "mov choice".NO[15] := NOT "space7";
       "mov choice".NO[16] := NOT "space11";
       "mov choice".NO[17] := NOT "space4";
       "mov choice".NO[18] := NOT "space8";
       "mov choice".NO[19] := NOT "space12"; // houseware import
       FOR "mov choice".i := 0 TO 19 DO
           IF "mov choice".NO["mov choice".i] THEN
               "X_coordinate" := "Locat"."shelf  X axis"["mov choice".i];
               "Y_coordinate" := "Locat"."shelf  Y axis"["mov choice".i];
               "Warehouse vacancies" := 1;
               "warn_NOspace(In.mod)" := 0;
               EXIT;
           ELSIF NOT "mov choice".NO["mov choice".i] THEN
               "X_coordinate" :=0;
               "Y_coordinate" :=0.0;
               "Warehouse vacancies" := 0;
               "warn_NOspace(In.mod)" := 1;
           END_IF;
           // Statement section FOR


       END_FOR;

   END_IF;
END_REGION

REGION Network 2 (SCL): 出库路径选择自动方案
   IF "outmod" THEN
       "mov choice".NO[0] := "space13"AND"mov_to13" ;
       "mov choice".NO[1] := "space17"AND"mov_to17";
       "mov choice".NO[2] := "space14" AND "mov_to14";
       "mov choice".NO[3] := "space18" AND "mov_to18";
       "mov choice".NO[4] := "space1" AND "mov_to1";
       "mov choice".NO[5] := "space5" AND "mov_to5";
       "mov choice".NO[6] := "space9" AND"mov_to9";
       "mov choice".NO[7] := "space15" AND"mov_to15";
       "mov choice".NO[8] := "space19" AND"mov_to19";
       "mov choice".NO[9] := "space2" AND"mov_to2";
       "mov choice".NO[10] := "space6" AND"mov_to6";
       "mov choice".NO[11] := "space10" AND"mov_to10";
       "mov choice".NO[12] := "space16" AND"mov_to16";
       "mov choice".NO[13] := "space20" AND"mov_to20";
       "mov choice".NO[14] := "space3" AND"mov_to3";
       "mov choice".NO[15] := "space7" AND"mov_to7";
       "mov choice".NO[16] := "space11" AND"mov_to11";
       "mov choice".NO[17] := "space4" AND"mov_to4";
       "mov choice".NO[18] := "space8" AND "mov_to8";
       "mov choice".NO[19] := "space12" AND"mov_to12"; // houseware export
       FOR "mov choice".i := 0 TO 19 DO
           IF "mov choice".NO["mov choice".i] THEN
               "X_coordinate" := "Locat"."shelf  X axis"["mov choice".i];
               "Y_coordinate" := "Locat"."shelf  Y axis"["mov choice".i];
               "outgoodsexist" := 1;
               EXIT;
           ELSIF NOT "mov choice".NO["mov choice".i] THEN
               "X_coordinate" := 0;
               "Y_coordinate" := 0.0;
               "outgoodsexist" := 0;
           END_IF;
           // Statement section FOR


       END_FOR;
   END_IF;
END_REGION
END_FUNCTION

FUNCTION "Y-axis stepper motor subroutine" : Void   // FC8, LAD
{ S7_Optimized_Access := 'TRUE' }
VERSION : 0.1
   VAR_TEMP   // added for the SCL form of the ladder/FBD networks
      _w1 : Bool;
   END_VAR
BEGIN

REGION Network 1
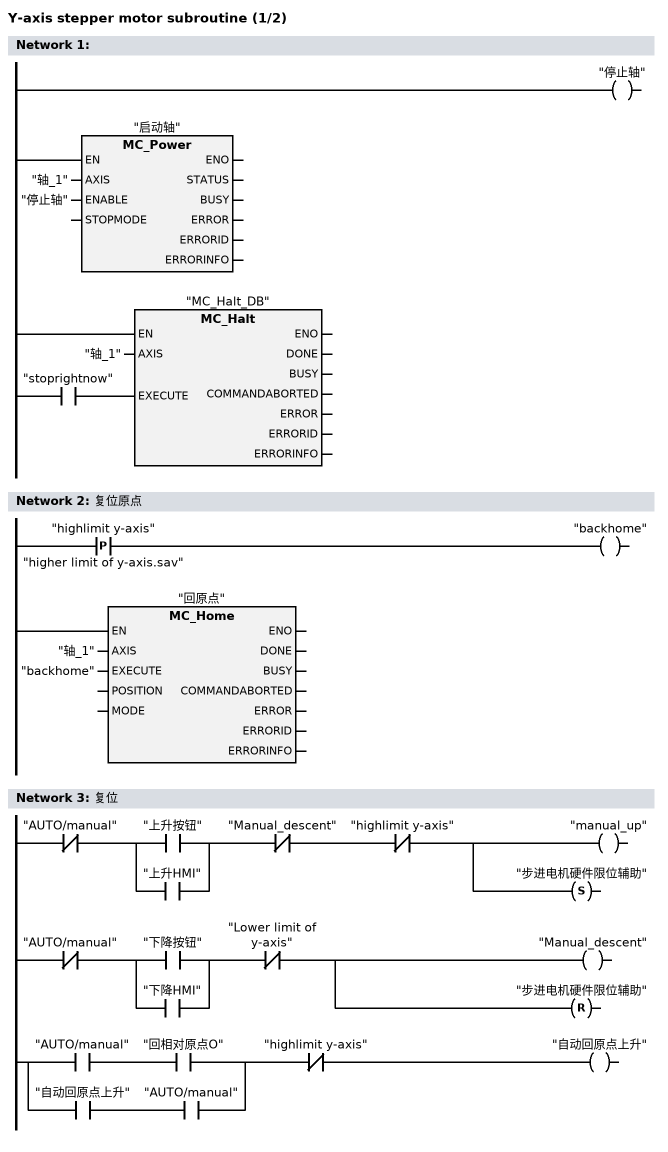
   "停止轴" := TRUE;
   "启动轴"(Axis := "轴_1", Enable := "停止轴");   // MC_Power
   "MC_Halt_DB"(Axis := "轴_1", Execute := "stoprightnow");   // MC_Halt
END_REGION

REGION Network 2: 复位原点
   #_w1 := "highlimit y-axis" AND NOT "higher limit of y-axis.sav";   // rising edge of "highlimit y-axis"
   "higher limit of y-axis.sav" := "highlimit y-axis";
   "backhome" := #_w1;
   "回原点"(Axis := "轴_1", Execute := "backhome");   // MC_Home
END_REGION

REGION Network 3: 复位
   RUNG wire#powerrail
      I_Contact( "AUTO/manual" )
      wire#w1
      Contact( "上升按钮" )
      wire#w2
      I_Contact( "Manual_descent" )
      I_Contact( "highlimit y-axis" )
      wire#w3
      Coil( "manual_up" )
   END_RUNG
   RUNG wire#w1
      Contact( "上升HMI" )
   END_RUNG wire#w2
   RUNG wire#w3
      S_Coil( "步进电机硬件限位辅助" )
   END_RUNG
   RUNG wire#powerrail
      I_Contact( "AUTO/manual" )
      wire#w4
      Contact( "下降按钮" )
      wire#w5
      I_Contact( "Lower limit of y-axis" )
      wire#w6
      Coil( "Manual_descent" )
   END_RUNG
   RUNG wire#w4
      Contact( "下降HMI" )
   END_RUNG wire#w5
   RUNG wire#w6
      R_Coil( "步进电机硬件限位辅助" )
   END_RUNG
   RUNG wire#powerrail
      Contact( "AUTO/manual" )
      Contact( "回相对原点O" )
      wire#w7
      I_Contact( "highlimit y-axis" )
      Coil( "自动回原点上升" )
   END_RUNG
   RUNG wire#powerrail
      Contact( "自动回原点上升" )
      Contact( "AUTO/manual" )
   END_RUNG wire#w7
   // the same network as SCL:
   "manual_up" := NOT "AUTO/manual" AND ("上升按钮" OR "上升HMI") AND NOT "Manual_descent" AND NOT "highlimit y-axis";
   IF "manual_up" THEN "步进电机硬件限位辅助" := TRUE; END_IF;
   "Manual_descent" := NOT "AUTO/manual" AND ("下降按钮" OR "下降HMI") AND NOT "Lower limit of y-axis";
   IF "Manual_descent" THEN "步进电机硬件限位辅助" := FALSE; END_IF;
   "自动回原点上升" := (("AUTO/manual" AND "回相对原点O") OR ("自动回原点上升" AND "AUTO/manual")) AND NOT "highlimit y-axis";
END_REGION

REGION Network 4: 手动
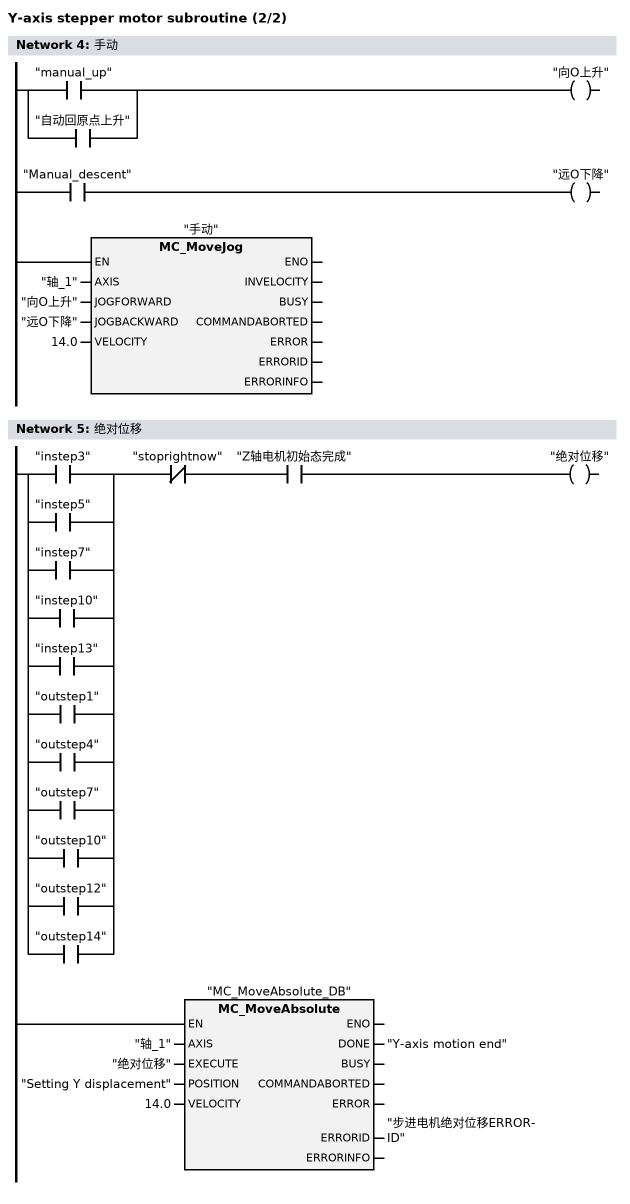
   "向O上升" := "manual_up" OR "自动回原点上升";
   "远O下降" := "Manual_descent";
   "手动"(Axis := "轴_1", JogForward := "向O上升", JogBackward := "远O下降", Velocity := 14.0);   // MC_MoveJog
END_REGION

REGION Network 5: 绝对位移
   "绝对位移" := ("instep3" OR "instep5" OR "instep7" OR "instep10" OR "instep13" OR "outstep1" OR "outstep4" OR "outstep7" OR "outstep10" OR "outstep12" OR "outstep14") AND NOT "stoprightnow" AND "Z轴电机初始态完成";
   "MC_MoveAbsolute_DB"(Axis := "轴_1",   // MC_MoveAbsolute
                        Execute := "绝对位移",
                        Position := "Setting Y displacement",
                        Velocity := 14.0,
                        Done => "Y-axis motion end",
                        ErrorID => "步进电机绝对位移ERROR-ID");
END_REGION
END_FUNCTION

FUNCTION "X-axis motor encoder group subroutine" : Void   // FC9, LAD
{ S7_Optimized_Access := 'TRUE' }
VERSION : 0.1
BEGIN

REGION Network 1
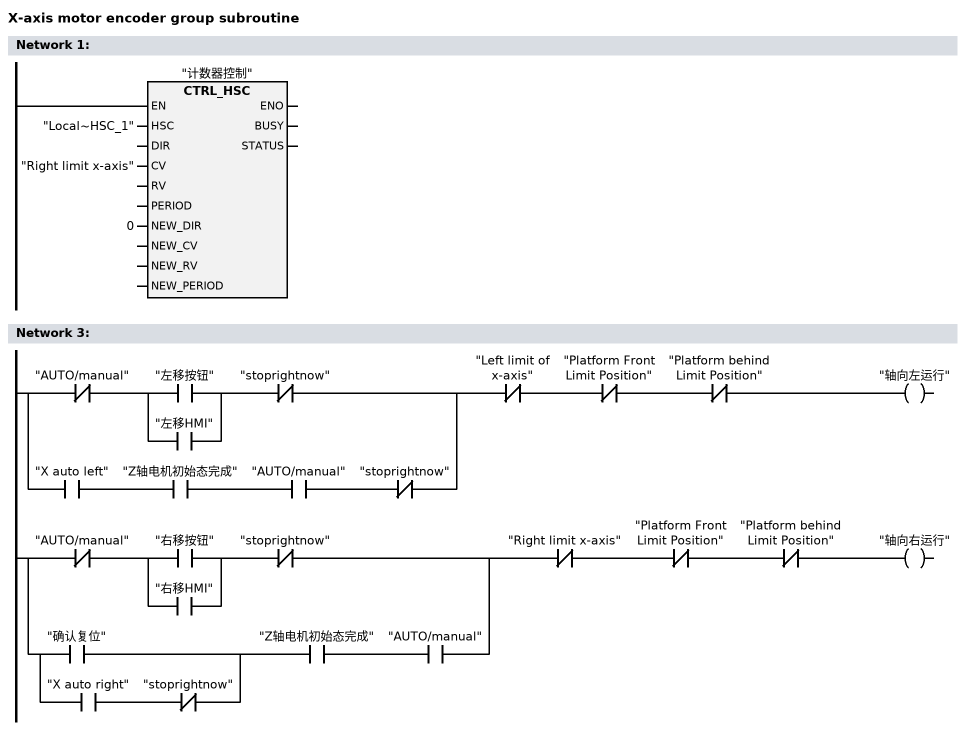
   "计数器控制"(HSC := "Local~HSC_1", CV := "Right limit x-axis", NEW_DIR := 0);   // CTRL_HSC
END_REGION

REGION Network 2 (SCL)
   //入库步序3-X轴
   IF ("instep3"OR "instep7"OR "outstep1"OR "outstep10") AND( "X-axis motion end"=0 ) THEN
       IF ("Pulse A-encoder value" < ("Setting X displacement" - 2)) AND (NOT "轴向右运行") THEN
           "X auto left" := 1;
           "X-axis right motion lock" := 1;
       ELSIF ("Pulse A-encoder value" > ("Setting X displacement" + 2)) AND (NOT "轴向左运行") THEN
           "X auto right" := 1;
           "X-axis left motion lock" := 1;
       END_IF;

       IF ("Pulse A-encoder value">=("Setting X displacement"-2))AND("X-axis left motion lock"=0)  THEN
           "X auto left" := 0;
           "X-axis motion end" := 1;
       ELSIF ("Pulse A-encoder value"<=("Setting X displacement"+2))AND("X-axis right motion lock"=0) THEN
       "X auto right":=0;
       "X-axis motion end" := 1;
   END_IF;

   END_IF;
END_REGION

REGION Network 3
   RUNG wire#powerrail
      I_Contact( "AUTO/manual" )
      wire#w1
      Contact( "左移按钮" )
      wire#w2
      I_Contact( "stoprightnow" )
      wire#w3
      I_Contact( "Left limit of x-axis" )
      I_Contact( "Platform Front Limit Position" )
      I_Contact( "Platform behind Limit Position" )
      Coil( "轴向左运行" )
   END_RUNG
   RUNG wire#w1
      Contact( "左移HMI" )
   END_RUNG wire#w2
   RUNG wire#powerrail
      Contact( "X auto left" )
      Contact( "Z轴电机初始态完成" )
      Contact( "AUTO/manual" )
      I_Contact( "stoprightnow" )
   END_RUNG wire#w3
   RUNG wire#powerrail
      I_Contact( "AUTO/manual" )
      wire#w4
      Contact( "右移按钮" )
      wire#w5
      I_Contact( "stoprightnow" )
      wire#w6
      I_Contact( "Right limit x-axis" )
      I_Contact( "Platform Front Limit Position" )
      I_Contact( "Platform behind Limit Position" )
      Coil( "轴向右运行" )
   END_RUNG
   RUNG wire#w4
      Contact( "右移HMI" )
   END_RUNG wire#w5
   RUNG wire#powerrail
      Contact( "确认复位" )
      wire#w7
      Contact( "Z轴电机初始态完成" )
      Contact( "AUTO/manual" )
   END_RUNG wire#w6
   RUNG wire#powerrail
      Contact( "X auto right" )
      I_Contact( "stoprightnow" )
   END_RUNG wire#w7
   // the same network as SCL:
   "轴向左运行" := ((NOT "AUTO/manual" AND ("左移按钮" OR "左移HMI") AND NOT "stoprightnow") OR ("X auto left" AND "Z轴电机初始态完成" AND "AUTO/manual" AND NOT "stoprightnow")) AND NOT "Left limit of x-axis" AND NOT "Platform Front Limit Position" AND NOT "Platform behind Limit Position";
   "轴向右运行" := ((NOT "AUTO/manual" AND ("右移按钮" OR "右移HMI") AND NOT "stoprightnow") OR (("确认复位" OR ("X auto right" AND NOT "stoprightnow")) AND "Z轴电机初始态完成" AND "AUTO/manual")) AND NOT "Right limit x-axis" AND NOT "Platform Front Limit Position" AND NOT "Platform behind Limit Position";
END_REGION
END_FUNCTION

FUNCTION "Z-axis motor subroutine" : Void   // FC10, LAD
{ S7_Optimized_Access := 'TRUE' }
VERSION : 0.1
   VAR_TEMP   // added for the SCL form of the ladder/FBD networks
      _w1 : Bool;
      _w2 : Bool;
   END_VAR
BEGIN

REGION Network 1: 去极限位
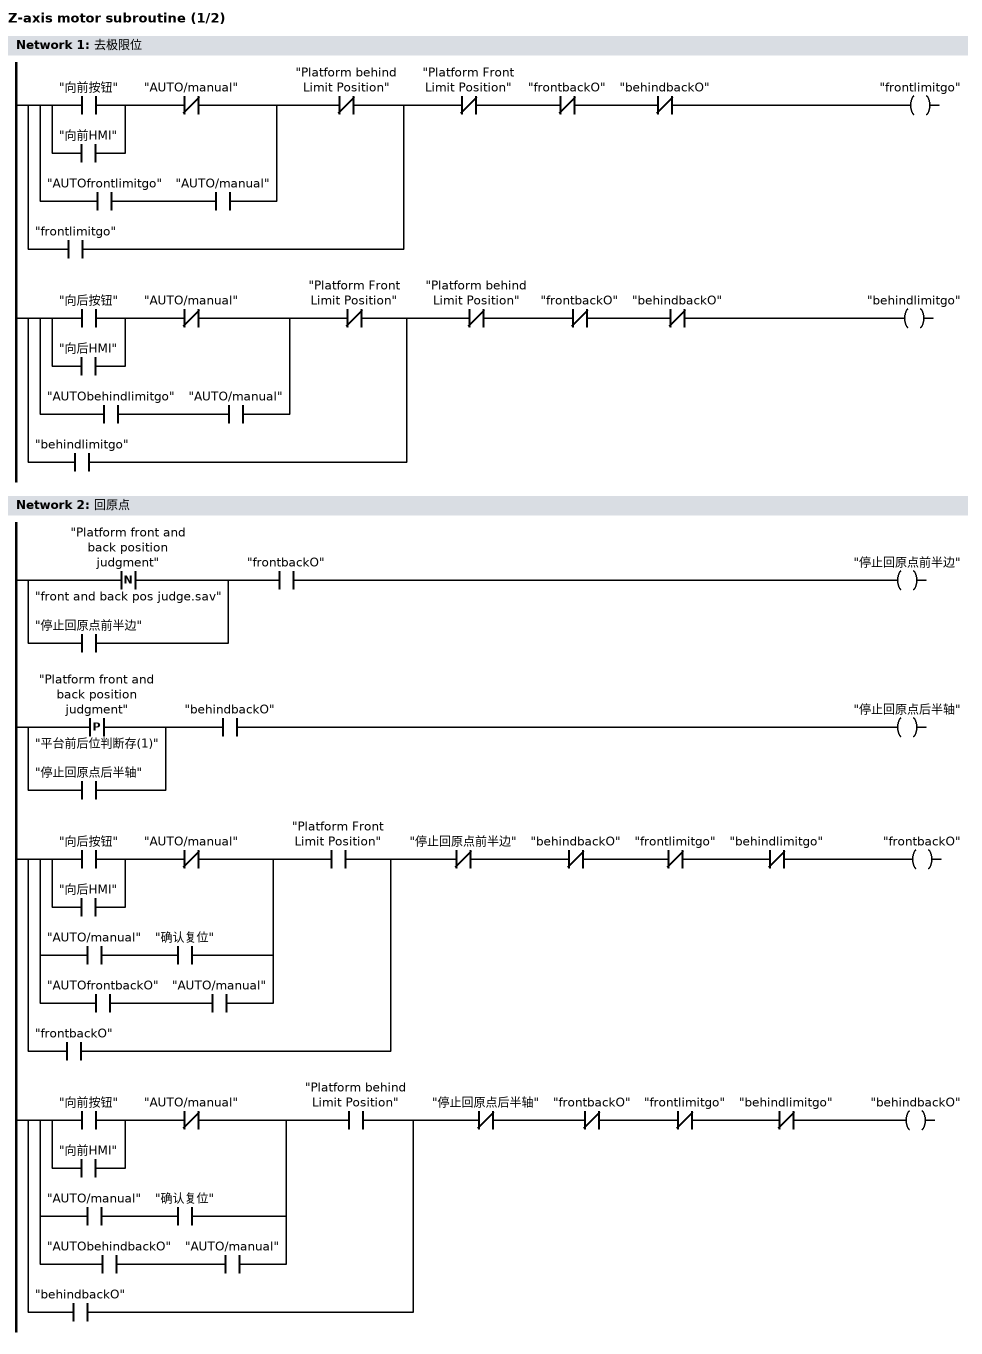
   RUNG wire#powerrail
      Contact( "向前按钮" )
      wire#w1
      I_Contact( "AUTO/manual" )
      wire#w2
      I_Contact( "Platform behind Limit Position" )
      wire#w3
      I_Contact( "Platform Front Limit Position" )
      I_Contact( "frontbackO" )
      I_Contact( "behindbackO" )
      Coil( "frontlimitgo" )
   END_RUNG
   RUNG wire#powerrail
      Contact( "向前HMI" )
   END_RUNG wire#w1
   RUNG wire#powerrail
      Contact( "AUTOfrontlimitgo" )
      Contact( "AUTO/manual" )
   END_RUNG wire#w2
   RUNG wire#powerrail
      Contact( "frontlimitgo" )
   END_RUNG wire#w3
   RUNG wire#powerrail
      Contact( "向后按钮" )
      wire#w4
      I_Contact( "AUTO/manual" )
      wire#w5
      I_Contact( "Platform Front Limit Position" )
      wire#w6
      I_Contact( "Platform behind Limit Position" )
      I_Contact( "frontbackO" )
      I_Contact( "behindbackO" )
      Coil( "behindlimitgo" )
   END_RUNG
   RUNG wire#powerrail
      Contact( "向后HMI" )
   END_RUNG wire#w4
   RUNG wire#powerrail
      Contact( "AUTObehindlimitgo" )
      Contact( "AUTO/manual" )
   END_RUNG wire#w5
   RUNG wire#powerrail
      Contact( "behindlimitgo" )
   END_RUNG wire#w6
   // the same network as SCL:
   "frontlimitgo" := ((((("向前按钮" OR "向前HMI") AND NOT "AUTO/manual") OR ("AUTOfrontlimitgo" AND "AUTO/manual")) AND NOT "Platform behind Limit Position") OR "frontlimitgo") AND NOT "Platform Front Limit Position" AND NOT "frontbackO" AND NOT "behindbackO";
   "behindlimitgo" := ((((("向后按钮" OR "向后HMI") AND NOT "AUTO/manual") OR ("AUTObehindlimitgo" AND "AUTO/manual")) AND NOT "Platform Front Limit Position") OR "behindlimitgo") AND NOT "Platform behind Limit Position" AND NOT "frontbackO" AND NOT "behindbackO";
END_REGION

REGION Network 2: 回原点
   RUNG wire#powerrail
      N_Contact(operand := "Platform front and back position judgment", bit := "front and back pos judge.sav")
      wire#w1
      Contact( "frontbackO" )
      Coil( "停止回原点前半边" )
   END_RUNG
   RUNG wire#powerrail
      Contact( "停止回原点前半边" )
   END_RUNG wire#w1
   RUNG wire#powerrail
      P_Contact(operand := "Platform front and back position judgment", bit := "平台前后位判断存(1)")
      wire#w2
      Contact( "behindbackO" )
      Coil( "停止回原点后半轴" )
   END_RUNG
   RUNG wire#powerrail
      Contact( "停止回原点后半轴" )
   END_RUNG wire#w2
   RUNG wire#powerrail
      Contact( "向后按钮" )
      wire#w3
      I_Contact( "AUTO/manual" )
      wire#w4
      Contact( "Platform Front Limit Position" )
      wire#w5
      I_Contact( "停止回原点前半边" )
      I_Contact( "behindbackO" )
      I_Contact( "frontlimitgo" )
      I_Contact( "behindlimitgo" )
      Coil( "frontbackO" )
   END_RUNG
   RUNG wire#powerrail
      Contact( "向后HMI" )
   END_RUNG wire#w3
   RUNG wire#powerrail
      Contact( "AUTO/manual" )
      Contact( "确认复位" )
   END_RUNG wire#w4
   RUNG wire#powerrail
      Contact( "AUTOfrontbackO" )
      Contact( "AUTO/manual" )
   END_RUNG wire#w4
   RUNG wire#powerrail
      Contact( "frontbackO" )
   END_RUNG wire#w5
   RUNG wire#powerrail
      Contact( "向前按钮" )
      wire#w6
      I_Contact( "AUTO/manual" )
      wire#w7
      Contact( "Platform behind Limit Position" )
      wire#w8
      I_Contact( "停止回原点后半轴" )
      I_Contact( "frontbackO" )
      I_Contact( "frontlimitgo" )
      I_Contact( "behindlimitgo" )
      Coil( "behindbackO" )
   END_RUNG
   RUNG wire#powerrail
      Contact( "向前HMI" )
   END_RUNG wire#w6
   RUNG wire#powerrail
      Contact( "AUTO/manual" )
      Contact( "确认复位" )
   END_RUNG wire#w7
   RUNG wire#powerrail
      Contact( "AUTObehindbackO" )
      Contact( "AUTO/manual" )
   END_RUNG wire#w7
   RUNG wire#powerrail
      Contact( "behindbackO" )
   END_RUNG wire#w8
   // the same network as SCL:
   #_w1 := NOT "Platform front and back position judgment" AND "front and back pos judge.sav";   // falling edge of "Platform front and back position judgment"
   "front and back pos judge.sav" := "Platform front and back position judgment";
   "停止回原点前半边" := (#_w1 OR "停止回原点前半边") AND "frontbackO";
   #_w2 := "Platform front and back position judgment" AND NOT "平台前后位判断存(1)";   // rising edge of "Platform front and back position judgment"
   "平台前后位判断存(1)" := "Platform front and back position judgment";
   "停止回原点后半轴" := (#_w2 OR "停止回原点后半轴") AND "behindbackO";
   "frontbackO" := ((((("向后按钮" OR "向后HMI") AND NOT "AUTO/manual") OR ("AUTO/manual" AND "确认复位") OR ("AUTOfrontbackO" AND "AUTO/manual")) AND "Platform Front Limit Position") OR "frontbackO") AND NOT "停止回原点前半边" AND NOT "behindbackO" AND NOT "frontlimitgo" AND NOT "behindlimitgo";
   "behindbackO" := ((((("向前按钮" OR "向前HMI") AND NOT "AUTO/manual") OR ("AUTO/manual" AND "确认复位") OR ("AUTObehindbackO" AND "AUTO/manual")) AND "Platform behind Limit Position") OR "behindbackO") AND NOT "停止回原点后半轴" AND NOT "frontbackO" AND NOT "frontlimitgo" AND NOT "behindlimitgo";
END_REGION

REGION Network 3: 电机控制段
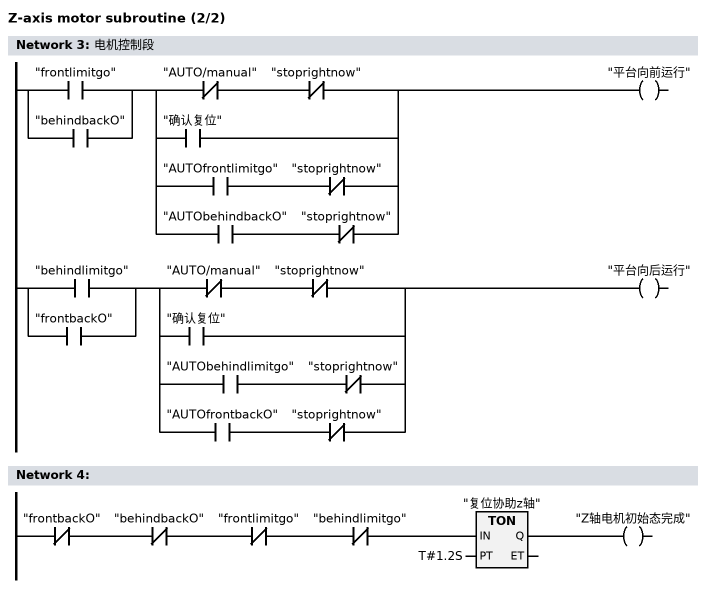
   RUNG wire#powerrail
      Contact( "frontlimitgo" )
      wire#w1
      I_Contact( "AUTO/manual" )
      I_Contact( "stoprightnow" )
      wire#w2
      Coil( "平台向前运行" )
   END_RUNG
   RUNG wire#powerrail
      Contact( "behindbackO" )
   END_RUNG wire#w1
   RUNG wire#w1
      Contact( "确认复位" )
   END_RUNG wire#w2
   RUNG wire#w1
      Contact( "AUTOfrontlimitgo" )
      I_Contact( "stoprightnow" )
   END_RUNG wire#w2
   RUNG wire#w1
      Contact( "AUTObehindbackO" )
      I_Contact( "stoprightnow" )
   END_RUNG wire#w2
   RUNG wire#powerrail
      Contact( "behindlimitgo" )
      wire#w3
      I_Contact( "AUTO/manual" )
      I_Contact( "stoprightnow" )
      wire#w4
      Coil( "平台向后运行" )
   END_RUNG
   RUNG wire#powerrail
      Contact( "frontbackO" )
   END_RUNG wire#w3
   RUNG wire#w3
      Contact( "确认复位" )
   END_RUNG wire#w4
   RUNG wire#w3
      Contact( "AUTObehindlimitgo" )
      I_Contact( "stoprightnow" )
   END_RUNG wire#w4
   RUNG wire#w3
      Contact( "AUTOfrontbackO" )
      I_Contact( "stoprightnow" )
   END_RUNG wire#w4
   // the same network as SCL:
   "平台向前运行" := ("frontlimitgo" OR "behindbackO") AND ((NOT "AUTO/manual" AND NOT "stoprightnow") OR "确认复位" OR ("AUTOfrontlimitgo" AND NOT "stoprightnow") OR ("AUTObehindbackO" AND NOT "stoprightnow"));
   "平台向后运行" := ("behindlimitgo" OR "frontbackO") AND ((NOT "AUTO/manual" AND NOT "stoprightnow") OR "确认复位" OR ("AUTObehindlimitgo" AND NOT "stoprightnow") OR ("AUTOfrontbackO" AND NOT "stoprightnow"));
END_REGION

REGION Network 4
   "复位协助z轴".TON(IN := NOT "frontbackO" AND NOT "behindbackO" AND NOT "frontlimitgo" AND NOT "behindlimitgo",
                PT := T#1.2S);
   "Z轴电机初始态完成" := "复位协助z轴".Q;
END_REGION
END_FUNCTION

FUNCTION "Warehouse scanning program" : Void   // FC11, LAD
{ S7_Optimized_Access := 'TRUE' }
VERSION : 0.1
BEGIN

REGION Network 1
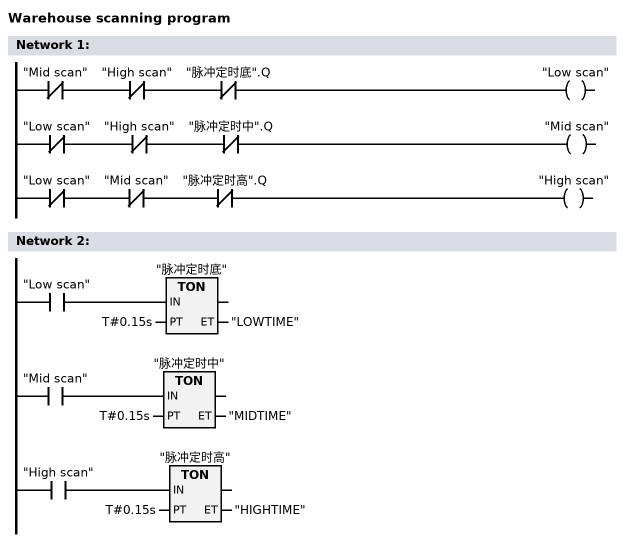
   RUNG wire#powerrail
      I_Contact( "Mid scan" )
      I_Contact( "High scan" )
      I_Contact( "脉冲定时底".Q )
      Coil( "Low scan" )
   END_RUNG
   RUNG wire#powerrail
      I_Contact( "Low scan" )
      I_Contact( "High scan" )
      I_Contact( "脉冲定时中".Q )
      Coil( "Mid scan" )
   END_RUNG
   RUNG wire#powerrail
      I_Contact( "Low scan" )
      I_Contact( "Mid scan" )
      I_Contact( "脉冲定时高".Q )
      Coil( "High scan" )
   END_RUNG
   // the same network as SCL:
   "Low scan" := NOT "Mid scan" AND NOT "High scan" AND NOT "脉冲定时底".Q;
   "Mid scan" := NOT "Low scan" AND NOT "High scan" AND NOT "脉冲定时中".Q;
   "High scan" := NOT "Low scan" AND NOT "Mid scan" AND NOT "脉冲定时高".Q;
END_REGION

REGION Network 2
   "脉冲定时底".TON(IN := "Low scan", PT := T#0.15s, ET => "LOWTIME");
   "脉冲定时中".TON(IN := "Mid scan", PT := T#0.15s, ET => "MIDTIME");
   "脉冲定时高".TON(IN := "High scan", PT := T#0.15s, ET => "HIGHTIME");
END_REGION

REGION Network 3 (SCL): 仓口1
   IF "Low scan" AND (("LOWTIME" > T#0.05s) AND ("LOWTIME" < T#0.1s)) THEN

       //货架1.NO1底层
       "space1" := NOT ("Low scan" = 1 AND "1.space in" = 0);
       "space2" := NOT ("Low scan" = 1 AND "2.space in" = 0);
       "space3" := NOT ("Low scan" = 1 AND "3.space in" = 0);
       "space4" := NOT ("Low scan" = 1 AND "4.space in" = 0);
       //货架2底层
       "space13" := NOT ("Low scan" = 1 AND "13.space in" = 0);
       "space14" := NOT ("Low scan" = 1 AND "14.space in" = 0);
       "space15" := NOT ("Low scan" = 1 AND "15.space in" = 0);
       "space16" := NOT ("Low scan" = 1 AND "16.space in" = 0);
   END_IF;

   IF "Mid scan"AND (("MIDTIME">T#0.05s)AND ("MIDTIME"<T#0.1s) )THEN
       //货架1.NO1中层
       "space5" := NOT ("Mid scan" = 1 AND "1.space in" = 0);
       "space6" := NOT ("Mid scan" = 1 AND "2.space in" = 0);
       "space7" := NOT ("Mid scan" = 1 AND "3.space in" = 0);
       "space8" := NOT ("Mid scan" = 1 AND "4.space in" = 0);
       //货架2中层
       "space17" := NOT ("Mid scan" = 1 AND "13.space in" = 0);
       "space18" := NOT ("Mid scan" = 1 AND "14.space in" = 0);
       "space19" := NOT ("Mid scan" = 1 AND "15.space in" = 0);
       "space20" := NOT ("Mid scan" = 1 AND "16.space in" = 0);
   END_IF;
   IF "High scan"AND (("HIGHTIME">T#0.05s)AND ("HIGHTIME"<T#0.1s) )THEN
       //货架1.NO2高层
       "space9" := NOT ("High scan" = 1 AND "1.space in" = 0);
       "space10" := NOT ("High scan" = 1 AND "2.space in" = 0);
       "space11" := NOT ("High scan" = 1 AND "3.space in" = 0);
       "space12" := NOT ("High scan" = 1 AND "4.space in" = 0);
       ;
   END_IF;
END_REGION
END_FUNCTION

FUNCTION "stop" : Void   // FC12, LAD
{ S7_Optimized_Access := 'TRUE' }
VERSION : 0.1
BEGIN

REGION Network 1 (SCL)
   "outmod" := 0;
   "inmod" := 0;
   "Z-axis motor subroutine"();
   "进货台逆时针" := 0;
   "进货台顺时针" := 0;
   "进货台电机驱动" := 0;
   "出货台顺时针" := 0;
   "出货台逆时针" := 0;
   "出货台电机驱动" := 0;
   "manual_up" := 0;
   "Manual_descent" := 0;
   "Y-axis stepper motor subroutine"();
   "进货台逆时针" :=0;
   "出货台顺时针" :=0;
   "X-axis motor encoder group subroutine"();
END_REGION
END_FUNCTION

FUNCTION "Auto in_ware Main Program" : Void   // FC13, SCL
{ S7_Optimized_Access := 'TRUE' }
VERSION : 0.1
BEGIN
   "Shelf Path Selection Subroutine"();//必须进入入库模式才可以访问本页面
   IF "inrequests" = 1 AND "inover" = 1 AND "insteps.sav" = 0 AND "Warehouse vacancies" AND "outrequests"=0  THEN
       "insteps.sav" := 1;
       "inover" := 0;
   END_IF;
   CASE "insteps.sav" OF
           // 取货步     
       1:"instep1" := 1;
       2:"instep2" := 1;
       3: "instep3" := 1;
           "in_Pick Pos Completion" := "X-axis motion end" AND "Y-axis motion end";
       4:"instep4" := 1;
       5:"instep5" := 1;
       6:"instep6" := 1;
           // 置货步   
       7:"instep7" := 1;
           "in_Pick Pos Completion" := "X-axis motion end" AND "Y-axis motion end";
       8:
           "instep8" := 1;
       9:"instep9" := 1;//调试原为"入库步序9" := 1
       10:"instep10" := 1;
       11:"instep11" := 1;
       12:
           "instep12" := 1;//调试原为"入库步序12" := 1
       13:"instep13" := 1;
       14:"instep14" := 1;
       15:"instep15" := 1;
       ELSE
           "insteps.sav" := 0; // 步序复位
           "inover" := 1;
   END_CASE;
   //开始取货
   //入库步序1
   IF "instep1" AND ("Incoming goods in place detection" = 0) THEN
       "进货台电机驱动" := 1 AND ("stoprightnow" = 0);
   ELSIF "instep1" AND ("Incoming goods in place detection" = 1) THEN
       "进货台电机驱动" := 0;
       "instep1" := 0;
       "insteps.sav" := "insteps.sav" + 1;
   END_IF;
   //入库步序2
   IF "instep2" AND ("enter table limit position" = 0) THEN
       "进货台顺时针" := 1 AND ("stoprightnow" = 0);
   ELSIF "instep2" AND ("enter table limit position" = 1) THEN
       "进货台顺时针" := 0;
       "instep2" := 0;
       "insteps.sav" := "insteps.sav" + 1;
   END_IF;
   //入库步序3

   IF "instep3" AND ("in_Pick Pos Completion" = 0) THEN
       "Z-axis motor subroutine"();
       IF "endLOCAT.X" >= 1360 AND "endLOCAT.Y"=-278.0 THEN
           "Setting Y displacement" := -278;
           "Y-axis stepper motor subroutine"();
           "X-axis motion end" := 1;//定位在同位
       ELSIF"endLOCAT.X" >= 1360 AND "endLOCAT.Y"=-145.0 THEN
           "Setting Y displacement" := -278;
           "Y-axis stepper motor subroutine"();
           "X-axis motion end" := 1;
       ELSIF NOT ("endLOCAT.X" >= 1360 )THEN
           "Setting X displacement" := 1362;
           "Setting Y displacement" := -278;
           "X-axis motor encoder group subroutine"();
           "Y-axis stepper motor subroutine"();
       END_IF;
   ELSIF "instep3" AND ("in_Pick Pos Completion" = 1) THEN
       "instep3" := 0;
       "insteps.sav" := "insteps.sav" + 1;
       "Setting Y displacement" := -120;
       "Y-axis stepper motor subroutine"();
       "X-axis motion end" := 0;
       "X-axis left motion lock" := 0;
       "X-axis right motion lock" := 0;
     "Setting X displacement" := 0;

   END_IF;
   //入库步序4
   IF "instep4" AND ("Platform behind Limit Position" = 0) THEN
       "AUTObehindlimitgo" := 1;
       "Z-axis motor subroutine"();
   ELSIF "instep4" AND ("Platform behind Limit Position" = 1) THEN
       "AUTObehindlimitgo" := 0;
       "instep4" := 0;
       "insteps.sav" := "insteps.sav" + 1;
   END_IF;
   //入库步序5
   IF "instep5" AND ("Y-axis motion end" = 0) THEN
       "Z-axis motor subroutine"();
       "Setting Y displacement" := -260;
       "Y-axis stepper motor subroutine"();
   ELSIF "instep5" AND ("Y-axis motion end" = 1) THEN
       "instep5" := 0;
       "insteps.sav" := "insteps.sav" + 1;
       "Setting Y displacement" := -120;
       "Y-axis stepper motor subroutine"();
   END_IF;
   //入库步序6
   IF "instep6" AND ("Platform behind Limit Position" = 1 OR "behindbackO" = 1) THEN
       "AUTObehindbackO" := 1;
       "Z-axis motor subroutine"();
   ELSIF "instep6" AND ("Platform behind Limit Position" = 0 AND "behindbackO" = 0) THEN
       "AUTObehindbackO" := 0;
       "instep6" := 0;
       "insteps.sav" := "insteps.sav" + 1;

   END_IF;
   //开始置货
   //入库步序7
   "time_scan_houseware".TP(IN := "instep7",
                            PT := T#0.4s,
                            Q => "Tscan_over",
                            ET => "Tscan_ET");
   IF "instep7" AND ("in_Pick Pos Completion" = 0) AND NOT "Tscan_over" THEN
       "Z-axis motor subroutine"();
       IF ("inset_running" = 0) OR( "WillLOCAT.X" = "X_coordinate"AND "WillLOCAT.Y" = ("Y_coordinate" - 15.0))  THEN
           IF "X_coordinate" = 1362 AND "Y_coordinate" = -263 THEN
               "Setting Y displacement" := -260.0;
               "Y-axis stepper motor subroutine"();
               "X-axis motion end" := 1;
               "WillLOCAT.X" := "X_coordinate";
               "WillLOCAT.Y" := ("Y_coordinate" - 15.0);
               "inset_running" := 1;
           ELSIF "X_coordinate" = 1362 AND "Y_coordinate" = -130 THEN
               "Setting Y displacement" := "Y_coordinate";
               "Y-axis stepper motor subroutine"();
               "X-axis motion end" := 1;
               "WillLOCAT.X" := "X_coordinate";
               "WillLOCAT.Y" := ("Y_coordinate" - 15.0);
               "inset_running" := 1;
           ELSE
               "Setting X displacement" := "X_coordinate";
               "Setting Y displacement" := "Y_coordinate";
               "X-axis motor encoder group subroutine"();
               "Y-axis stepper motor subroutine"();
               "WillLOCAT.X" := "X_coordinate";
               "WillLOCAT.Y" := ("Y_coordinate" - 15.0);
               "inset_running" := 1;
           END_IF;// Statement section IF
       ELSE
           "stoprightnow" := 1;
           "error_spacewrong(In.mod)" := 1;
       END_IF;

   ELSIF "instep7" AND ("in_Pick Pos Completion" = 1) THEN
       "instep7" := 0;
       "insteps.sav" := "insteps.sav" + 1;
       "Setting Y displacement" := -120;
       "Y-axis stepper motor subroutine"();
       "X-axis motion end" := 0;
       "X-axis left motion lock" := 0;
       "X-axis right motion lock" := 0;
       "Setting X displacement" := 0;
       "endLOCAT.X" := "X_coordinate";
       "endLOCAT.Y" := ("Y_coordinate" - 15.0);
       "inset_running" := 0;
       "mov choice".WZ := "mov choice".i;
   END_IF;
   //入库步序8
   IF "instep8" THEN
       IF     "WillLOCAT.X" = "X_coordinate"AND "WillLOCAT.Y" = ("Y_coordinate" - 15.0) THEN
           IF "X_coordinate" = 929 OR "X_coordinate" = 633 OR "X_coordinate" = 334 OR "X_coordinate" = 34 THEN
               "instep8" := 0;
               "insteps.sav" := "insteps.sav" + 1;
           ELSIF "X_coordinate" = 1362 OR "X_coordinate" = 1061 OR "X_coordinate" = 764 OR "X_coordinate" = 466 THEN
               "instep8" := 0;
               "insteps.sav" := "insteps.sav" + 4;
               ;
           END_IF;  // Statement section IF// Statement section IF
       ELSE
           "stoprightnow" := 1;
           "error_spacewrong(In.mod)" := 1;
       END_IF;



   END_IF;

       //置入货架1
       //入库步序9
       IF "instep9" AND ("Platform behind Limit Position" = 0) THEN
           "AUTObehindlimitgo" := 1;
           "Z-axis motor subroutine"();
       ELSIF "instep9" AND ("Platform behind Limit Position" = 1) THEN
           "AUTObehindlimitgo" := 0;
           "instep9" := 0;
           "insteps.sav" := "insteps.sav" + 1;
       END_IF;
       //入库步序10
       IF "instep10" AND ("Y-axis motion end" = 0) THEN
           "Z-axis motor subroutine"();
               "Setting Y displacement" := ("Y_coordinate" - 15.0);
               "Y-axis stepper motor subroutine"();
       ELSIF "instep10" AND ("Y-axis motion end" = 1) THEN
           "instep10" := 0;
           "insteps.sav" := "insteps.sav" + 1;
           "Setting Y displacement" := -120;
           "Y-axis stepper motor subroutine"();
       END_IF;
       //入库步序11
       IF "instep11" AND ("Platform behind Limit Position" = 1 OR "behindbackO" = 1) THEN
           "AUTObehindbackO" := 1;
           "Z-axis motor subroutine"();
       ELSIF "instep11" AND ("Platform behind Limit Position" = 0 AND "behindbackO" = 0) THEN
           "AUTObehindbackO" := 0;
           "instep11" := 0;
           "insteps.sav" := "insteps.sav" + 4;
       END_IF;
       //置入货架2
       //入库步序12
       IF "instep12" AND ("Platform Front Limit Position" = 0) THEN
           "AUTOfrontlimitgo" := 1;
           "Z-axis motor subroutine"();
       ELSIF "instep12" AND ("Platform Front Limit Position" = 1) THEN
           "AUTOfrontlimitgo" := 0;
           "instep12" := 0;
           "insteps.sav" := "insteps.sav" + 1;
       END_IF;
       //入库步序13
       IF "instep13" AND ("Y-axis motion end" = 0) THEN
           "Z-axis motor subroutine"();
               "Setting Y displacement" := ("Y_coordinate" - 15.0);
               "Y-axis stepper motor subroutine"();
       ELSIF "instep13" AND ("Y-axis motion end" = 1) THEN
           "instep13" := 0;
           "insteps.sav" := "insteps.sav" + 1;
           "Setting Y displacement" := -120;
           "Y-axis stepper motor subroutine"();
       END_IF;
       //入库步序14
       IF "instep14" AND ("Platform Front Limit Position" = 1 OR "frontbackO" = 1) THEN
           "AUTOfrontbackO" := 1;
           "Z-axis motor subroutine"();
       ELSIF "instep14" AND ("Platform Front Limit Position" = 0 AND "frontbackO" = 0) THEN
           "AUTOfrontbackO" := 0;
           "instep14" := 0;
           "insteps.sav" := "insteps.sav" + 1;
       END_IF;

   //入库步序15进货台归位
   IF "instep15" AND ("enter table Zero position" = 0) THEN
       "进货台逆时针" := 1 AND ("stoprightnow" = 0);
       "error_goodslose(IN.mod)" := ("instep15" AND "mov choice".NO["mov choice".WZ]);
       "stoprightnow" := "error_goodslose(IN.mod)";
   ELSIF "instep15" AND ("enter table Zero position" = 1)AND "mov choice".NO["mov choice".WZ]=0 THEN
       "进货台逆时针" := 0;
       "instep15" := 0;
       "WillLOCAT.X" := 0;
       "WillLOCAT.Y" := 0;
       "mov choice".WZ := 0;
       "insteps.sav":="insteps.sav" + 1;//原为"顺控步序":="顺控步序" + 1
   END_IF;
END_FUNCTION

ORGANIZATION_BLOCK "Main"   // OB1, LAD, ProgramCycle
TITLE = "Main Program Sweep (Cycle)"
{ S7_Optimized_Access := 'TRUE' }
VERSION : 0.1
BEGIN

REGION Network 1
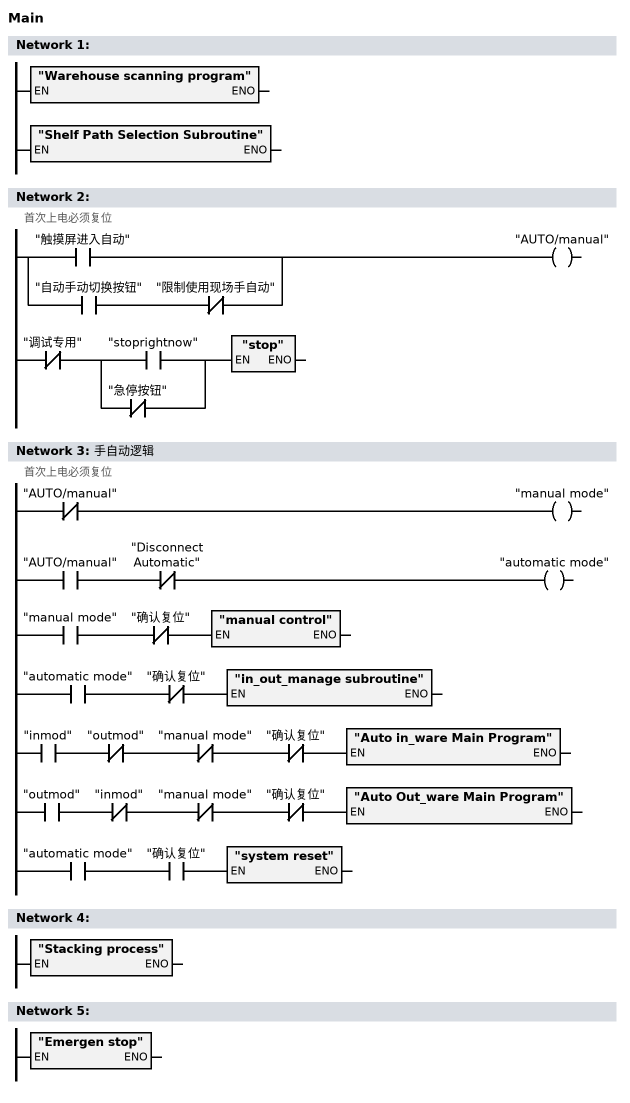
   RUNG wire#powerrail
      "Warehouse scanning program"()
   END_RUNG
   RUNG wire#powerrail
      "Shelf Path Selection Subroutine"()
   END_RUNG
   // the same network as SCL:
   "Warehouse scanning program"();
   "Shelf Path Selection Subroutine"();
END_REGION

REGION Network 2
   // 首次上电必须复位
   RUNG wire#powerrail
      Contact( "触摸屏进入自动" )
      wire#w1
      Coil( "AUTO/manual" )
   END_RUNG
   RUNG wire#powerrail
      Contact( "自动手动切换按钮" )
      I_Contact( "限制使用现场手自动" )
   END_RUNG wire#w1
   RUNG wire#powerrail
      I_Contact( "调试专用" )
      wire#w2
      Contact( "stoprightnow" )
      wire#w3
      "stop"()
   END_RUNG
   RUNG wire#w2
      I_Contact( "急停按钮" )
   END_RUNG wire#w3
   // the same network as SCL:
   "AUTO/manual" := "触摸屏进入自动" OR ("自动手动切换按钮" AND NOT "限制使用现场手自动");
   IF NOT "调试专用" AND ("stoprightnow" OR NOT "急停按钮") THEN "stop"(); END_IF;
END_REGION

REGION Network 3: 手自动逻辑
   // 首次上电必须复位
   RUNG wire#powerrail
      I_Contact( "AUTO/manual" )
      Coil( "manual mode" )
   END_RUNG
   RUNG wire#powerrail
      Contact( "AUTO/manual" )
      I_Contact( "Disconnect Automatic" )
      Coil( "automatic mode" )
   END_RUNG
   RUNG wire#powerrail
      Contact( "manual mode" )
      I_Contact( "确认复位" )
      "manual control"()
   END_RUNG
   RUNG wire#powerrail
      Contact( "automatic mode" )
      I_Contact( "确认复位" )
      "in_out_manage subroutine"()
   END_RUNG
   RUNG wire#powerrail
      Contact( "inmod" )
      I_Contact( "outmod" )
      I_Contact( "manual mode" )
      I_Contact( "确认复位" )
      "Auto in_ware Main Program"()
   END_RUNG
   RUNG wire#powerrail
      Contact( "outmod" )
      I_Contact( "inmod" )
      I_Contact( "manual mode" )
      I_Contact( "确认复位" )
      "Auto Out_ware Main Program"()
   END_RUNG
   RUNG wire#powerrail
      Contact( "automatic mode" )
      Contact( "确认复位" )
      "system reset"()
   END_RUNG
   // the same network as SCL:
   "manual mode" := NOT "AUTO/manual";
   "automatic mode" := "AUTO/manual" AND NOT "Disconnect Automatic";
   IF "manual mode" AND NOT "确认复位" THEN "manual control"(); END_IF;
   IF "automatic mode" AND NOT "确认复位" THEN "in_out_manage subroutine"(); END_IF;
   IF "inmod" AND NOT "outmod" AND NOT "manual mode" AND NOT "确认复位" THEN
       "Auto in_ware Main Program"();
   END_IF;
   IF "outmod" AND NOT "inmod" AND NOT "manual mode" AND NOT "确认复位" THEN
       "Auto Out_ware Main Program"();
   END_IF;
   IF "automatic mode" AND "确认复位" THEN "system reset"(); END_IF;
END_REGION

REGION Network 4
   RUNG wire#powerrail
      "Stacking process"()
   END_RUNG
   // the same network as SCL:
   "Stacking process"();
END_REGION

REGION Network 5
   RUNG wire#powerrail
      "Emergen stop"()
   END_RUNG
   // the same network as SCL:
   "Emergen stop"();
END_REGION
END_ORGANIZATION_BLOCK

ORGANIZATION_BLOCK "Startup"   // OB100, LAD, Startup
TITLE = "Complete Restart"
{ S7_Optimized_Access := 'TRUE' }
VERSION : 0.1
   VAR_INPUT
      LostRetentive : Bool;   // True if retentive data are lost
      LostRTC : Bool;   // True if date and time are lost
   END_VAR
BEGIN

REGION Network 1
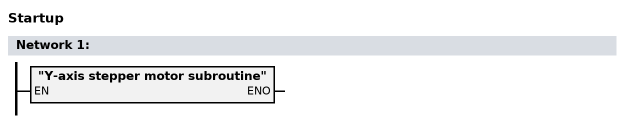
   RUNG wire#powerrail
      "Y-axis stepper motor subroutine"()
   END_RUNG
   // the same network as SCL:
   "Y-axis stepper motor subroutine"();
END_REGION
END_ORGANIZATION_BLOCK

// folder: 堆垛系统

FUNCTION "Stacking process" : Void   // FC4, LAD
{ S7_Optimized_Access := 'TRUE' }
VERSION : 0.1
   VAR_TEMP   // added for the SCL form of the ladder/FBD networks
      _w1 : Bool;
      _w2 : Bool;
      _w3 : Bool;
   END_VAR
BEGIN

REGION Network 1
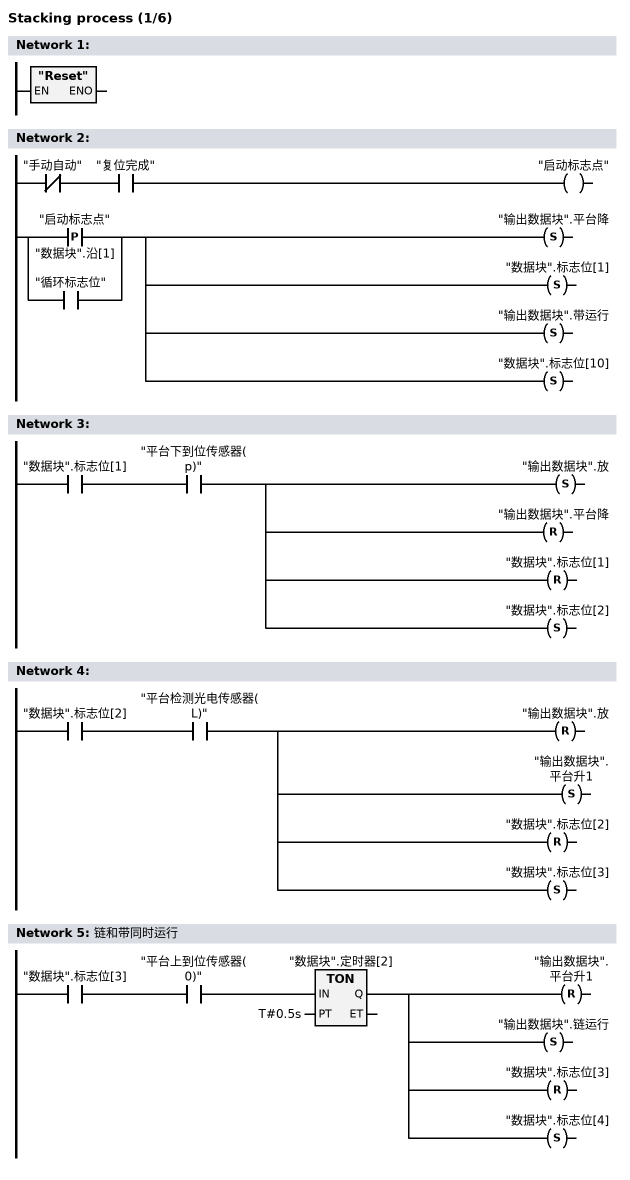
   RUNG wire#powerrail
      "Reset"()
   END_RUNG
   // the same network as SCL:
   "Reset"();
END_REGION

REGION Network 2
   RUNG wire#powerrail
      I_Contact( "手动自动" )
      Contact( "复位完成" )
      Coil( "启动标志点" )
   END_RUNG
   RUNG wire#powerrail
      P_Contact(operand := "启动标志点", bit := "数据块".沿[1])
      wire#w1
      S_Coil( "输出数据块".平台降 )
   END_RUNG
   RUNG wire#powerrail
      Contact( "循环标志位" )
   END_RUNG wire#w1
   RUNG wire#w1
      S_Coil( "数据块".标志位[1] )
   END_RUNG
   RUNG wire#w1
      S_Coil( "输出数据块".带运行 )
   END_RUNG
   RUNG wire#w1
      S_Coil( "数据块".标志位[10] )
   END_RUNG
   // the same network as SCL:
   "启动标志点" := NOT "手动自动" AND "复位完成";
   #_w1 := "启动标志点" AND NOT "数据块".沿[1];   // rising edge of "启动标志点"
   "数据块".沿[1] := "启动标志点";
   IF #_w1 OR "循环标志位" THEN
       "输出数据块".平台降 := TRUE;
       "数据块".标志位[1] := TRUE;
       "输出数据块".带运行 := TRUE;
       "数据块".标志位[10] := TRUE;
   END_IF;
END_REGION

REGION Network 3
   RUNG wire#powerrail
      Contact( "数据块".标志位[1] )
      Contact( "平台下到位传感器(p)" )
      wire#w1
      S_Coil( "输出数据块".放 )
   END_RUNG
   RUNG wire#w1
      R_Coil( "输出数据块".平台降 )
   END_RUNG
   RUNG wire#w1
      R_Coil( "数据块".标志位[1] )
   END_RUNG
   RUNG wire#w1
      S_Coil( "数据块".标志位[2] )
   END_RUNG
   // the same network as SCL:
   IF "数据块".标志位[1] AND "平台下到位传感器(p)" THEN
       "输出数据块".放 := TRUE;
       "输出数据块".平台降 := FALSE;
   END_IF;
   #_w1 := "数据块".标志位[1] AND "平台下到位传感器(p)";
   IF #_w1 THEN
       "数据块".标志位[1] := FALSE;
       "数据块".标志位[2] := TRUE;
   END_IF;
END_REGION

REGION Network 4
   RUNG wire#powerrail
      Contact( "数据块".标志位[2] )
      Contact( "平台检测光电传感器(L)" )
      wire#w1
      R_Coil( "输出数据块".放 )
   END_RUNG
   RUNG wire#w1
      S_Coil( "输出数据块".平台升1 )
   END_RUNG
   RUNG wire#w1
      R_Coil( "数据块".标志位[2] )
   END_RUNG
   RUNG wire#w1
      S_Coil( "数据块".标志位[3] )
   END_RUNG
   // the same network as SCL:
   IF "数据块".标志位[2] AND "平台检测光电传感器(L)" THEN
       "输出数据块".放 := FALSE;
       "输出数据块".平台升1 := TRUE;
   END_IF;
   #_w1 := "数据块".标志位[2] AND "平台检测光电传感器(L)";
   IF #_w1 THEN
       "数据块".标志位[2] := FALSE;
       "数据块".标志位[3] := TRUE;
   END_IF;
END_REGION

REGION Network 5: 链和带同时运行
   "数据块".定时器[2].TON(IN := "数据块".标志位[3] AND "平台上到位传感器(0)", PT := T#0.5s);
   IF "数据块".定时器[2].Q THEN
       "输出数据块".平台升1 := FALSE;
       "输出数据块".链运行 := TRUE;
       "数据块".标志位[3] := FALSE;
       "数据块".标志位[4] := TRUE;
   END_IF;
END_REGION

REGION Network 6
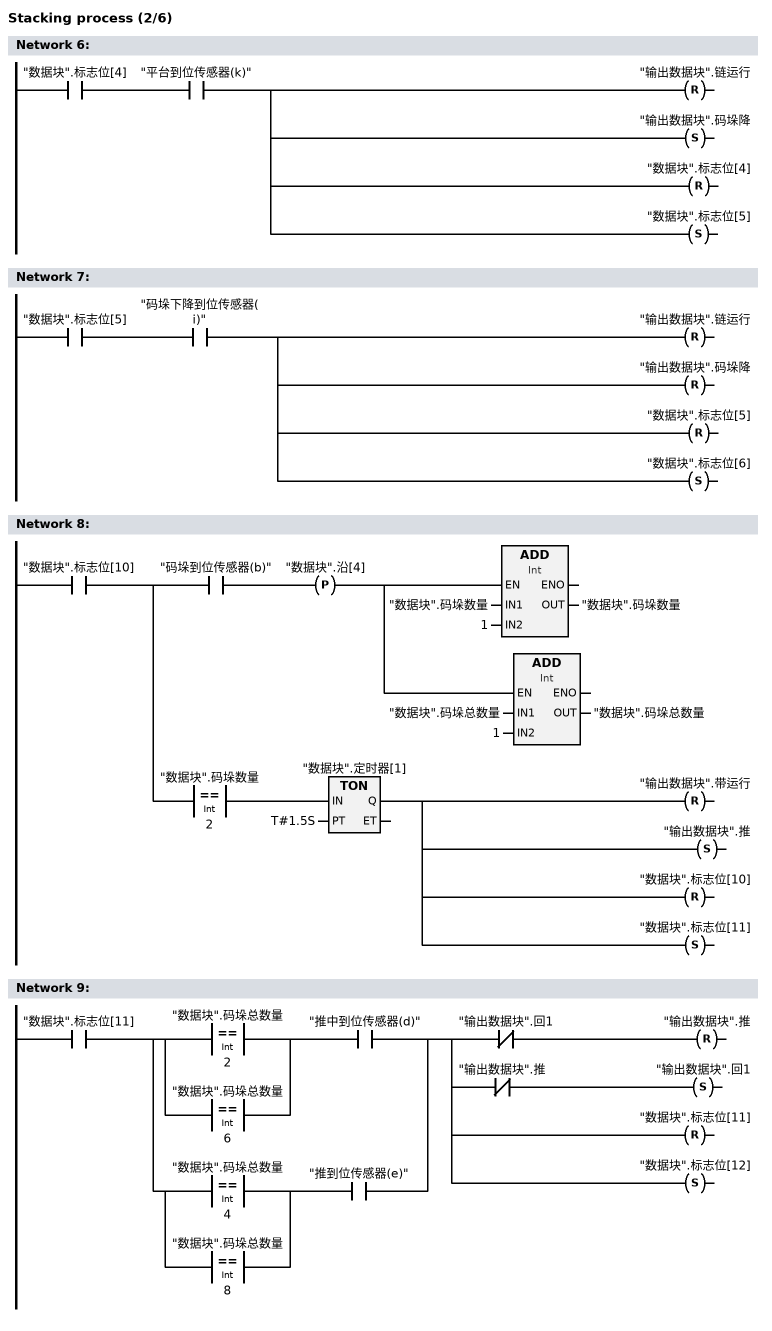
   RUNG wire#powerrail
      Contact( "数据块".标志位[4] )
      Contact( "平台到位传感器(k)" )
      wire#w1
      R_Coil( "输出数据块".链运行 )
   END_RUNG
   RUNG wire#w1
      S_Coil( "输出数据块".码垛降 )
   END_RUNG
   RUNG wire#w1
      R_Coil( "数据块".标志位[4] )
   END_RUNG
   RUNG wire#w1
      S_Coil( "数据块".标志位[5] )
   END_RUNG
   // the same network as SCL:
   IF "数据块".标志位[4] AND "平台到位传感器(k)" THEN
       "输出数据块".链运行 := FALSE;
       "输出数据块".码垛降 := TRUE;
   END_IF;
   #_w1 := "数据块".标志位[4] AND "平台到位传感器(k)";
   IF #_w1 THEN
       "数据块".标志位[4] := FALSE;
       "数据块".标志位[5] := TRUE;
   END_IF;
END_REGION

REGION Network 7
   RUNG wire#powerrail
      Contact( "数据块".标志位[5] )
      Contact( "码垛下降到位传感器(i)" )
      wire#w1
      R_Coil( "输出数据块".链运行 )
   END_RUNG
   RUNG wire#w1
      R_Coil( "输出数据块".码垛降 )
   END_RUNG
   RUNG wire#w1
      R_Coil( "数据块".标志位[5] )
   END_RUNG
   RUNG wire#w1
      S_Coil( "数据块".标志位[6] )
   END_RUNG
   // the same network as SCL:
   IF "数据块".标志位[5] AND "码垛下降到位传感器(i)" THEN
       "输出数据块".链运行 := FALSE;
       "输出数据块".码垛降 := FALSE;
   END_IF;
   #_w1 := "数据块".标志位[5] AND "码垛下降到位传感器(i)";
   IF #_w1 THEN
       "数据块".标志位[5] := FALSE;
       "数据块".标志位[6] := TRUE;
   END_IF;
END_REGION

REGION Network 8
   #_w1 := "数据块".标志位[10] AND "码垛到位传感器(b)";
   #_w2 := #_w1 AND NOT "数据块".沿[4];   // rising edge
   "数据块".沿[4] := #_w1;
   IF #_w2 THEN
       "数据块".码垛数量 := "数据块".码垛数量 + 1;
       "数据块".码垛总数量 := "数据块".码垛总数量 + 1;
   END_IF;
   "数据块".定时器[1].TON(IN := "数据块".标志位[10] AND ("数据块".码垛数量 = 2), PT := T#1.5S);
   IF "数据块".定时器[1].Q THEN
       "输出数据块".带运行 := FALSE;
       "输出数据块".推 := TRUE;
       "数据块".标志位[10] := FALSE;
       "数据块".标志位[11] := TRUE;
   END_IF;
END_REGION

REGION Network 9
   RUNG wire#powerrail
      Contact( "数据块".标志位[11] )
      wire#w1
      { S7_Templates := "SrcType := Int" } EQ_Contact(in1 := "数据块".码垛总数量, in2 := 2)
      wire#w2
      Contact( "推中到位传感器(d)" )
      wire#w3
      I_Contact( "输出数据块".回1 )
      R_Coil( "输出数据块".推 )
   END_RUNG
   RUNG wire#w1
      { S7_Templates := "SrcType := Int" } EQ_Contact(in1 := "数据块".码垛总数量, in2 := 6)
   END_RUNG wire#w2
   RUNG wire#w1
      { S7_Templates := "SrcType := Int" } EQ_Contact(in1 := "数据块".码垛总数量, in2 := 4)
      wire#w4
      Contact( "推到位传感器(e)" )
   END_RUNG wire#w3
   RUNG wire#w1
      { S7_Templates := "SrcType := Int" } EQ_Contact(in1 := "数据块".码垛总数量, in2 := 8)
   END_RUNG wire#w4
   RUNG wire#w3
      I_Contact( "输出数据块".推 )
      S_Coil( "输出数据块".回1 )
   END_RUNG
   RUNG wire#w3
      R_Coil( "数据块".标志位[11] )
   END_RUNG
   RUNG wire#w3
      S_Coil( "数据块".标志位[12] )
   END_RUNG
   // the same network as SCL:
   #_w1 := "数据块".标志位[11] AND (((("数据块".码垛总数量 = 2) OR ("数据块".码垛总数量 = 6)) AND "推中到位传感器(d)") OR ((("数据块".码垛总数量 = 4) OR ("数据块".码垛总数量 = 8)) AND "推到位传感器(e)"));
   IF #_w1 AND NOT "输出数据块".回1 THEN "输出数据块".推 := FALSE; END_IF;
   IF #_w1 AND NOT "输出数据块".推 THEN "输出数据块".回1 := TRUE; END_IF;
   IF #_w1 THEN
       "数据块".标志位[11] := FALSE;
       "数据块".标志位[12] := TRUE;
   END_IF;
END_REGION

REGION Network 10
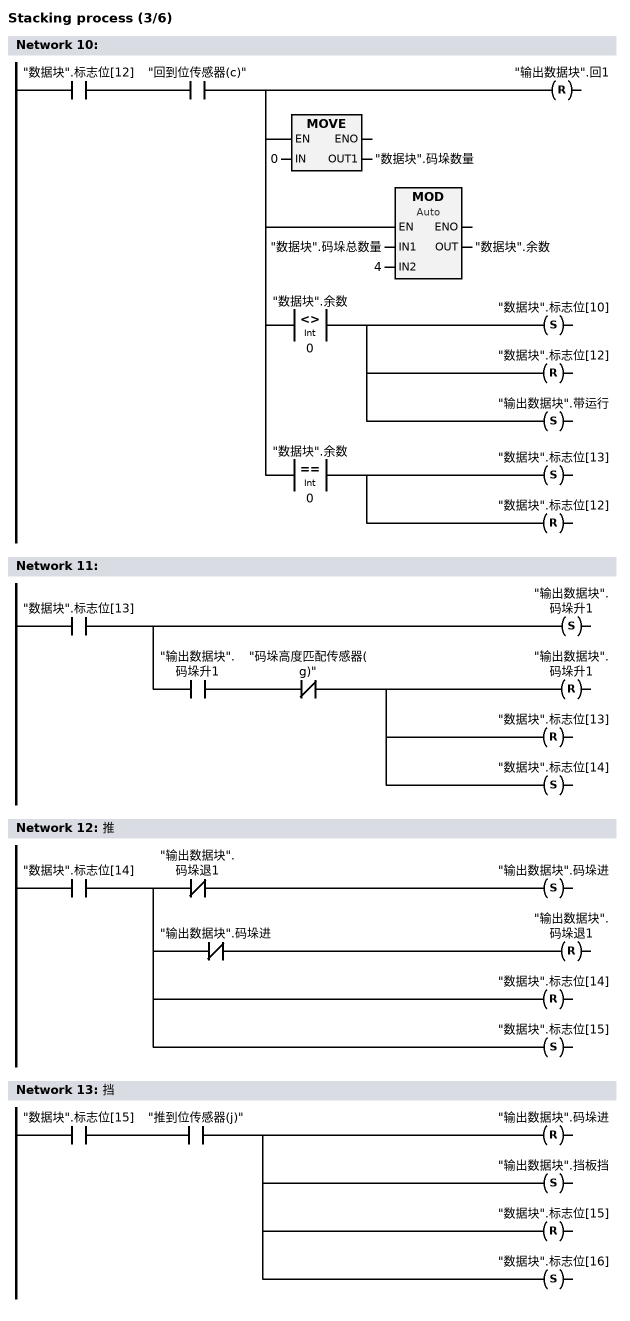
   RUNG wire#powerrail
      Contact( "数据块".标志位[12] )
      Contact( "回到位传感器(c)" )
      wire#w1
      R_Coil( "输出数据块".回1 )
   END_RUNG
   RUNG wire#w1
      { S7_GenerateENO := "TRUE" } Move(in := 0, out1 => "数据块".码垛数量)
   END_RUNG
   RUNG wire#w1
      { S7_GenerateENO := "TRUE" } Mod(in1 := "数据块".码垛总数量, in2 := 4, out => "数据块".余数)
   END_RUNG
   RUNG wire#w1
      { S7_Templates := "SrcType := Int" } NE_Contact(in1 := "数据块".余数, in2 := 0)
      wire#w2
      S_Coil( "数据块".标志位[10] )
   END_RUNG
   RUNG wire#w2
      R_Coil( "数据块".标志位[12] )
   END_RUNG
   RUNG wire#w2
      S_Coil( "输出数据块".带运行 )
   END_RUNG
   RUNG wire#w1
      { S7_Templates := "SrcType := Int" } EQ_Contact(in1 := "数据块".余数, in2 := 0)
      wire#w3
      S_Coil( "数据块".标志位[13] )
   END_RUNG
   RUNG wire#w3
      R_Coil( "数据块".标志位[12] )
   END_RUNG
   // the same network as SCL:
   #_w1 := "数据块".标志位[12] AND "回到位传感器(c)";
   IF #_w1 THEN
       "输出数据块".回1 := FALSE;
       "数据块".码垛数量 := 0;
       "数据块".余数 := "数据块".码垛总数量 MOD 4;
   END_IF;
   IF #_w1 AND ("数据块".余数 <> 0) THEN
       "数据块".标志位[10] := TRUE;
       "数据块".标志位[12] := FALSE;
       "输出数据块".带运行 := TRUE;
   END_IF;
   IF #_w1 AND ("数据块".余数 = 0) THEN
       "数据块".标志位[13] := TRUE;
       "数据块".标志位[12] := FALSE;
   END_IF;
END_REGION

REGION Network 11
   RUNG wire#powerrail
      Contact( "数据块".标志位[13] )
      wire#w1
      S_Coil( "输出数据块".码垛升1 )
   END_RUNG
   RUNG wire#w1
      Contact( "输出数据块".码垛升1 )
      I_Contact( "码垛高度匹配传感器(g)" )
      wire#w2
      R_Coil( "输出数据块".码垛升1 )
   END_RUNG
   RUNG wire#w2
      R_Coil( "数据块".标志位[13] )
   END_RUNG
   RUNG wire#w2
      S_Coil( "数据块".标志位[14] )
   END_RUNG
   // the same network as SCL:
   IF "数据块".标志位[13] THEN "输出数据块".码垛升1 := TRUE; END_IF;
   #_w1 := "数据块".标志位[13] AND "输出数据块".码垛升1 AND NOT "码垛高度匹配传感器(g)";
   IF #_w1 THEN
       "输出数据块".码垛升1 := FALSE;
       "数据块".标志位[13] := FALSE;
       "数据块".标志位[14] := TRUE;
   END_IF;
END_REGION

REGION Network 12: 推
   RUNG wire#powerrail
      Contact( "数据块".标志位[14] )
      wire#w1
      I_Contact( "输出数据块".码垛退1 )
      S_Coil( "输出数据块".码垛进 )
   END_RUNG
   RUNG wire#w1
      I_Contact( "输出数据块".码垛进 )
      R_Coil( "输出数据块".码垛退1 )
   END_RUNG
   RUNG wire#w1
      R_Coil( "数据块".标志位[14] )
   END_RUNG
   RUNG wire#w1
      S_Coil( "数据块".标志位[15] )
   END_RUNG
   // the same network as SCL:
   IF "数据块".标志位[14] AND NOT "输出数据块".码垛退1 THEN "输出数据块".码垛进 := TRUE; END_IF;
   IF "数据块".标志位[14] AND NOT "输出数据块".码垛进 THEN "输出数据块".码垛退1 := FALSE; END_IF;
   #_w1 := "数据块".标志位[14];
   IF #_w1 THEN
       "数据块".标志位[14] := FALSE;
       "数据块".标志位[15] := TRUE;
   END_IF;
END_REGION

REGION Network 13: 挡
   RUNG wire#powerrail
      Contact( "数据块".标志位[15] )
      Contact( "推到位传感器(j)" )
      wire#w1
      R_Coil( "输出数据块".码垛进 )
   END_RUNG
   RUNG wire#w1
      S_Coil( "输出数据块".挡板挡 )
   END_RUNG
   RUNG wire#w1
      R_Coil( "数据块".标志位[15] )
   END_RUNG
   RUNG wire#w1
      S_Coil( "数据块".标志位[16] )
   END_RUNG
   // the same network as SCL:
   IF "数据块".标志位[15] AND "推到位传感器(j)" THEN
       "输出数据块".码垛进 := FALSE;
       "输出数据块".挡板挡 := TRUE;
   END_IF;
   #_w1 := "数据块".标志位[15] AND "推到位传感器(j)";
   IF #_w1 THEN
       "数据块".标志位[15] := FALSE;
       "数据块".标志位[16] := TRUE;
   END_IF;
END_REGION

REGION Network 14
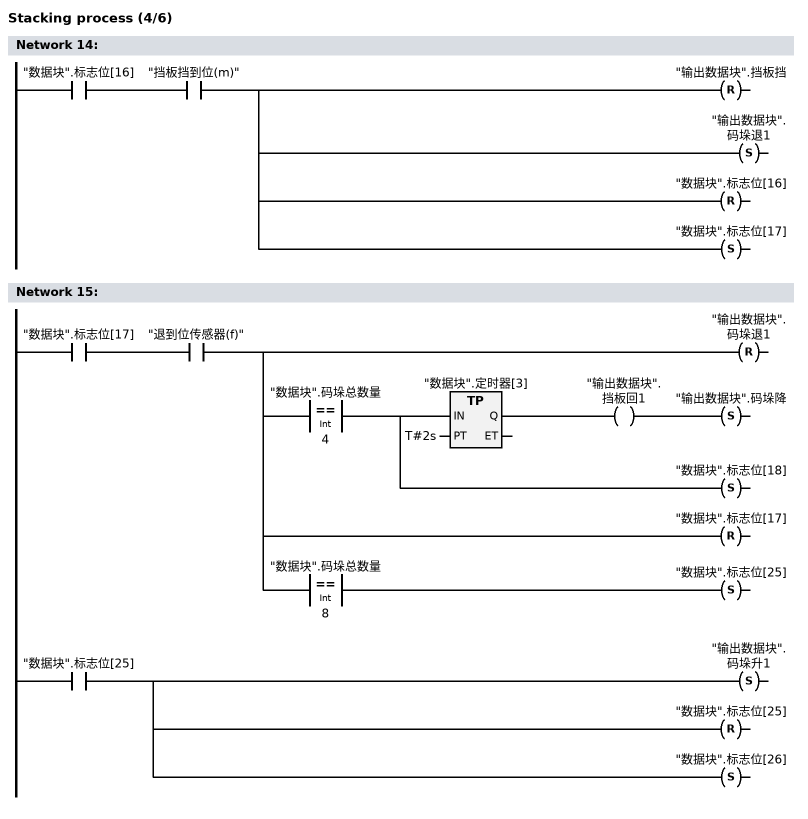
   RUNG wire#powerrail
      Contact( "数据块".标志位[16] )
      Contact( "挡板挡到位(m)" )
      wire#w1
      R_Coil( "输出数据块".挡板挡 )
   END_RUNG
   RUNG wire#w1
      S_Coil( "输出数据块".码垛退1 )
   END_RUNG
   RUNG wire#w1
      R_Coil( "数据块".标志位[16] )
   END_RUNG
   RUNG wire#w1
      S_Coil( "数据块".标志位[17] )
   END_RUNG
   // the same network as SCL:
   IF "数据块".标志位[16] AND "挡板挡到位(m)" THEN
       "输出数据块".挡板挡 := FALSE;
       "输出数据块".码垛退1 := TRUE;
   END_IF;
   #_w1 := "数据块".标志位[16] AND "挡板挡到位(m)";
   IF #_w1 THEN
       "数据块".标志位[16] := FALSE;
       "数据块".标志位[17] := TRUE;
   END_IF;
END_REGION

REGION Network 15
   #_w1 := "数据块".标志位[17] AND "退到位传感器(f)";
   IF #_w1 THEN "输出数据块".码垛退1 := FALSE; END_IF;
   #_w2 := #_w1 AND ("数据块".码垛总数量 = 4);
   "数据块".定时器[3].TP(IN := #_w2, PT := T#2s);
   "输出数据块".挡板回1 := "数据块".定时器[3].Q;
   IF "数据块".定时器[3].Q THEN "输出数据块".码垛降 := TRUE; END_IF;
   IF #_w2 THEN "数据块".标志位[18] := TRUE; END_IF;
   IF #_w1 THEN "数据块".标志位[17] := FALSE; END_IF;
   IF #_w1 AND ("数据块".码垛总数量 = 8) THEN "数据块".标志位[25] := TRUE; END_IF;
   IF "数据块".标志位[25] THEN "输出数据块".码垛升1 := TRUE; END_IF;
   #_w3 := "数据块".标志位[25];
   IF #_w3 THEN
       "数据块".标志位[25] := FALSE;
       "数据块".标志位[26] := TRUE;
   END_IF;
END_REGION

REGION Network 16
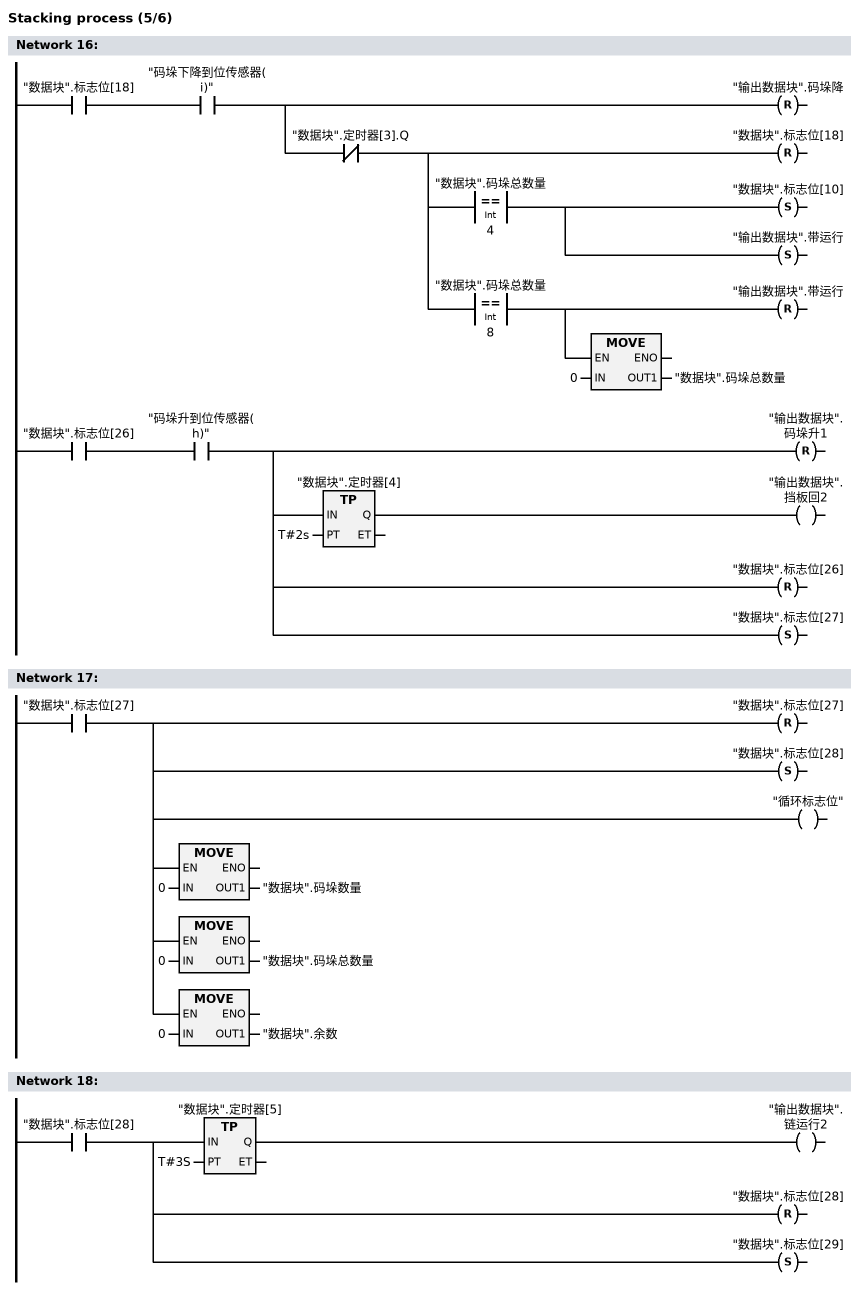
   #_w1 := "数据块".标志位[18] AND "码垛下降到位传感器(i)";
   IF #_w1 THEN "输出数据块".码垛降 := FALSE; END_IF;
   #_w2 := #_w1 AND NOT "数据块".定时器[3].Q;
   IF #_w2 THEN "数据块".标志位[18] := FALSE; END_IF;
   IF #_w2 AND ("数据块".码垛总数量 = 4) THEN
       "数据块".标志位[10] := TRUE;
       "输出数据块".带运行 := TRUE;
   END_IF;
   IF #_w2 AND ("数据块".码垛总数量 = 8) THEN
       "输出数据块".带运行 := FALSE;
       "数据块".码垛总数量 := 0;
   END_IF;
   #_w3 := "数据块".标志位[26] AND "码垛升到位传感器(h)";
   IF #_w3 THEN "输出数据块".码垛升1 := FALSE; END_IF;
   "数据块".定时器[4].TP(IN := #_w3, PT := T#2s);
   "输出数据块".挡板回2 := "数据块".定时器[4].Q;
   IF #_w3 THEN
       "数据块".标志位[26] := FALSE;
       "数据块".标志位[27] := TRUE;
   END_IF;
END_REGION

REGION Network 17
   RUNG wire#powerrail
      Contact( "数据块".标志位[27] )
      wire#w1
      R_Coil( "数据块".标志位[27] )
   END_RUNG
   RUNG wire#w1
      S_Coil( "数据块".标志位[28] )
   END_RUNG
   RUNG wire#w1
      Coil( "循环标志位" )
   END_RUNG
   RUNG wire#w1
      { S7_GenerateENO := "TRUE" } Move(in := 0, out1 => "数据块".码垛数量)
   END_RUNG
   RUNG wire#w1
      { S7_GenerateENO := "TRUE" } Move(in := 0, out1 => "数据块".码垛总数量)
   END_RUNG
   RUNG wire#w1
      { S7_GenerateENO := "TRUE" } Move(in := 0, out1 => "数据块".余数)
   END_RUNG
   // the same network as SCL:
   #_w1 := "数据块".标志位[27];
   IF #_w1 THEN
       "数据块".标志位[27] := FALSE;
       "数据块".标志位[28] := TRUE;
   END_IF;
   "循环标志位" := #_w1;
   IF #_w1 THEN
       "数据块".码垛数量 := 0;
       "数据块".码垛总数量 := 0;
       "数据块".余数 := 0;
   END_IF;
END_REGION

REGION Network 18
   "数据块".定时器[5].TP(IN := "数据块".标志位[28], PT := T#3S);
   "输出数据块".链运行2 := "数据块".定时器[5].Q;
   #_w1 := "数据块".标志位[28];
   IF #_w1 THEN
       "数据块".标志位[28] := FALSE;
       "数据块".标志位[29] := TRUE;
   END_IF;
END_REGION

REGION Network 19
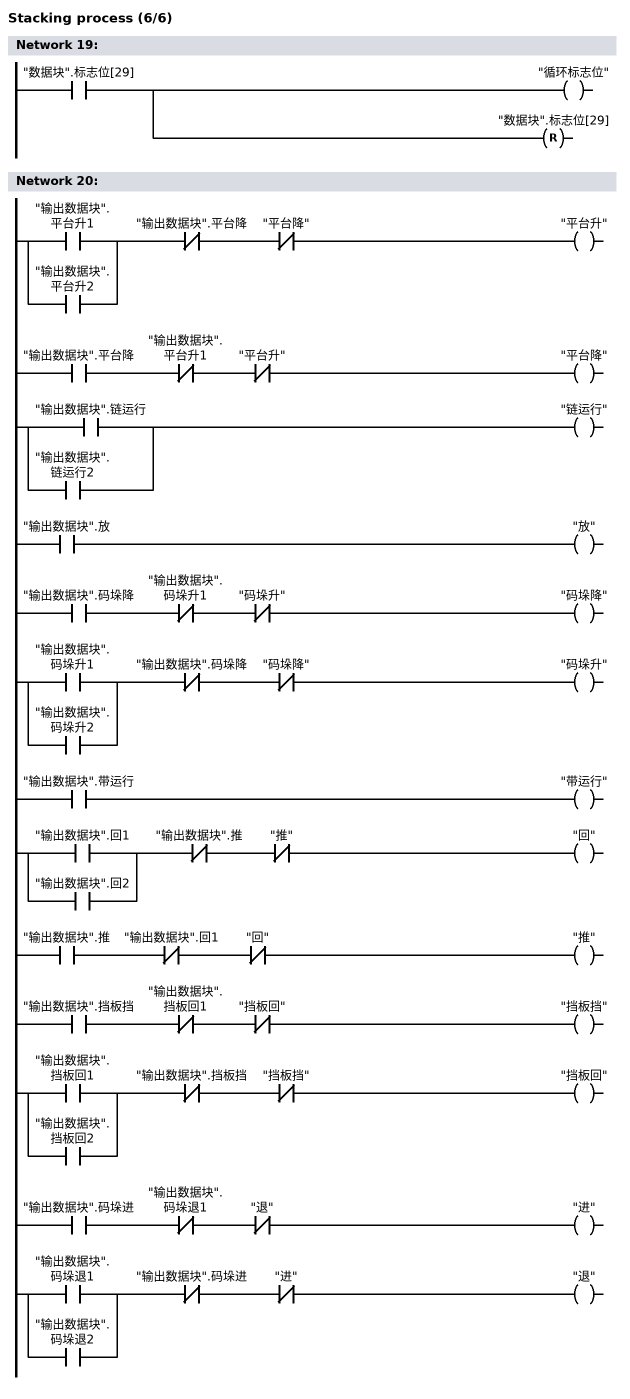
   RUNG wire#powerrail
      Contact( "数据块".标志位[29] )
      wire#w1
      Coil( "循环标志位" )
   END_RUNG
   RUNG wire#w1
      R_Coil( "数据块".标志位[29] )
   END_RUNG
   // the same network as SCL:
   "循环标志位" := "数据块".标志位[29];
   IF "数据块".标志位[29] THEN "数据块".标志位[29] := FALSE; END_IF;
END_REGION

REGION Network 20
   RUNG wire#powerrail
      Contact( "输出数据块".平台升1 )
      wire#w1
      I_Contact( "输出数据块".平台降 )
      I_Contact( "平台降" )
      Coil( "平台升" )
   END_RUNG
   RUNG wire#powerrail
      Contact( "输出数据块".平台升2 )
   END_RUNG wire#w1
   RUNG wire#powerrail
      Contact( "输出数据块".平台降 )
      I_Contact( "输出数据块".平台升1 )
      I_Contact( "平台升" )
      Coil( "平台降" )
   END_RUNG
   RUNG wire#powerrail
      Contact( "输出数据块".链运行 )
      wire#w2
      Coil( "链运行" )
   END_RUNG
   RUNG wire#powerrail
      Contact( "输出数据块".链运行2 )
   END_RUNG wire#w2
   RUNG wire#powerrail
      Contact( "输出数据块".放 )
      Coil( "放" )
   END_RUNG
   RUNG wire#powerrail
      Contact( "输出数据块".码垛降 )
      I_Contact( "输出数据块".码垛升1 )
      I_Contact( "码垛升" )
      Coil( "码垛降" )
   END_RUNG
   RUNG wire#powerrail
      Contact( "输出数据块".码垛升1 )
      wire#w3
      I_Contact( "输出数据块".码垛降 )
      I_Contact( "码垛降" )
      Coil( "码垛升" )
   END_RUNG
   RUNG wire#powerrail
      Contact( "输出数据块".码垛升2 )
   END_RUNG wire#w3
   RUNG wire#powerrail
      Contact( "输出数据块".带运行 )
      Coil( "带运行" )
   END_RUNG
   RUNG wire#powerrail
      Contact( "输出数据块".回1 )
      wire#w4
      I_Contact( "输出数据块".推 )
      I_Contact( "推" )
      Coil( "回" )
   END_RUNG
   RUNG wire#powerrail
      Contact( "输出数据块".回2 )
   END_RUNG wire#w4
   RUNG wire#powerrail
      Contact( "输出数据块".推 )
      I_Contact( "输出数据块".回1 )
      I_Contact( "回" )
      Coil( "推" )
   END_RUNG
   RUNG wire#powerrail
      Contact( "输出数据块".挡板挡 )
      I_Contact( "输出数据块".挡板回1 )
      I_Contact( "挡板回" )
      Coil( "挡板挡" )
   END_RUNG
   RUNG wire#powerrail
      Contact( "输出数据块".挡板回1 )
      wire#w5
      I_Contact( "输出数据块".挡板挡 )
      I_Contact( "挡板挡" )
      Coil( "挡板回" )
   END_RUNG
   RUNG wire#powerrail
      Contact( "输出数据块".挡板回2 )
   END_RUNG wire#w5
   RUNG wire#powerrail
      Contact( "输出数据块".码垛进 )
      I_Contact( "输出数据块".码垛退1 )
      I_Contact( "退" )
      Coil( "进" )
   END_RUNG
   RUNG wire#powerrail
      Contact( "输出数据块".码垛退1 )
      wire#w6
      I_Contact( "输出数据块".码垛进 )
      I_Contact( "进" )
      Coil( "退" )
   END_RUNG
   RUNG wire#powerrail
      Contact( "输出数据块".码垛退2 )
   END_RUNG wire#w6
   // the same network as SCL:
   "平台升" := ("输出数据块".平台升1 OR "输出数据块".平台升2) AND NOT "输出数据块".平台降 AND NOT "平台降";
   "平台降" := "输出数据块".平台降 AND NOT "输出数据块".平台升1 AND NOT "平台升";
   "链运行" := "输出数据块".链运行 OR "输出数据块".链运行2;
   "放" := "输出数据块".放;
   "码垛降" := "输出数据块".码垛降 AND NOT "输出数据块".码垛升1 AND NOT "码垛升";
   "码垛升" := ("输出数据块".码垛升1 OR "输出数据块".码垛升2) AND NOT "输出数据块".码垛降 AND NOT "码垛降";
   "带运行" := "输出数据块".带运行;
   "回" := ("输出数据块".回1 OR "输出数据块".回2) AND NOT "输出数据块".推 AND NOT "推";
   "推" := "输出数据块".推 AND NOT "输出数据块".回1 AND NOT "回";
   "挡板挡" := "输出数据块".挡板挡 AND NOT "输出数据块".挡板回1 AND NOT "挡板回";
   "挡板回" := ("输出数据块".挡板回1 OR "输出数据块".挡板回2) AND NOT "输出数据块".挡板挡 AND NOT "挡板挡";
   "进" := "输出数据块".码垛进 AND NOT "输出数据块".码垛退1 AND NOT "退";
   "退" := ("输出数据块".码垛退1 OR "输出数据块".码垛退2) AND NOT "输出数据块".码垛进 AND NOT "进";
END_REGION
END_FUNCTION

FUNCTION "Emergen stop" : Void   // FC14, LAD
{ S7_Optimized_Access := 'TRUE' }
VERSION : 0.1
   VAR_TEMP   // added for the SCL form of the ladder/FBD networks
      _w1 : Bool;
   END_VAR
BEGIN

REGION Network 2
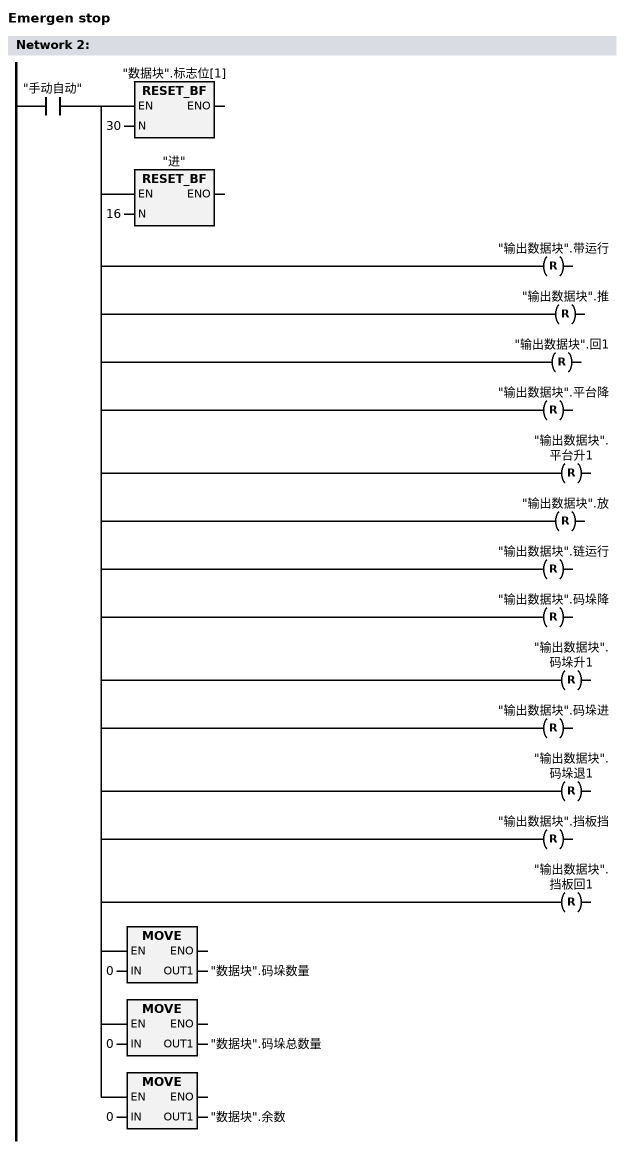
   // no SCL statement known for RBitfield: written as a call
   IF "手动自动" THEN RESET_BF(operand := "数据块".标志位[1], n := 30); END_IF;
   #_w1 := "手动自动";
   IF #_w1 THEN
       RESET_BF(operand := "进", n := 16);
       "输出数据块".带运行 := FALSE;
       "输出数据块".推 := FALSE;
       "输出数据块".回1 := FALSE;
       "输出数据块".平台降 := FALSE;
       "输出数据块".平台升1 := FALSE;
       "输出数据块".放 := FALSE;
       "输出数据块".链运行 := FALSE;
       "输出数据块".码垛降 := FALSE;
       "输出数据块".码垛升1 := FALSE;
       "输出数据块".码垛进 := FALSE;
       "输出数据块".码垛退1 := FALSE;
       "输出数据块".挡板挡 := FALSE;
       "输出数据块".挡板回1 := FALSE;
       "数据块".码垛数量 := 0;
       "数据块".码垛总数量 := 0;
       "数据块".余数 := 0;
   END_IF;
END_REGION
END_FUNCTION

FUNCTION "Reset" : Void   // FC15, LAD
{ S7_Optimized_Access := 'TRUE' }
VERSION : 0.1
   VAR_TEMP   // added for the SCL form of the ladder/FBD networks
      _w1 : Bool;
   END_VAR
BEGIN

REGION Network 1
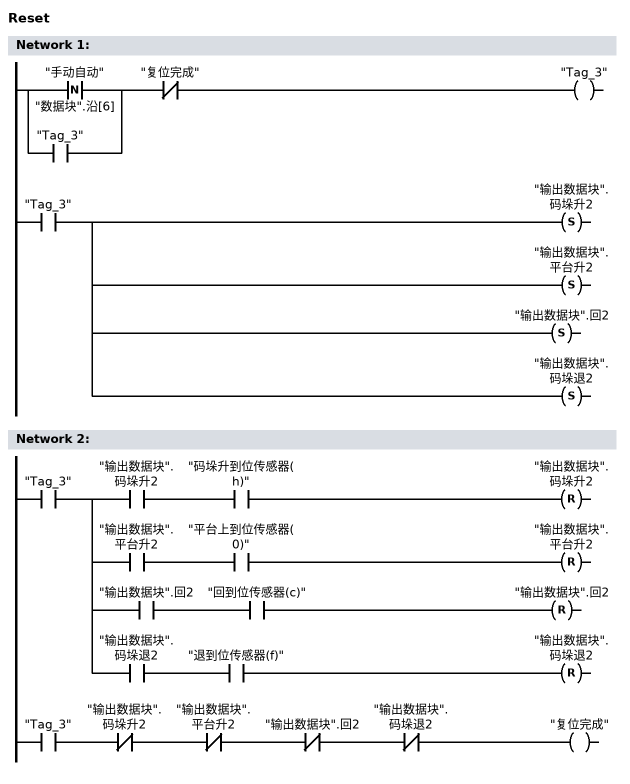
   RUNG wire#powerrail
      N_Contact(operand := "手动自动", bit := "数据块".沿[6])
      wire#w1
      I_Contact( "复位完成" )
      Coil( "Tag_3" )
   END_RUNG
   RUNG wire#powerrail
      Contact( "Tag_3" )
   END_RUNG wire#w1
   RUNG wire#powerrail
      Contact( "Tag_3" )
      wire#w2
      S_Coil( "输出数据块".码垛升2 )
   END_RUNG
   RUNG wire#w2
      S_Coil( "输出数据块".平台升2 )
   END_RUNG
   RUNG wire#w2
      S_Coil( "输出数据块".回2 )
   END_RUNG
   RUNG wire#w2
      S_Coil( "输出数据块".码垛退2 )
   END_RUNG
   // the same network as SCL:
   #_w1 := NOT "手动自动" AND "数据块".沿[6];   // falling edge of "手动自动"
   "数据块".沿[6] := "手动自动";
   "Tag_3" := (#_w1 OR "Tag_3") AND NOT "复位完成";
   IF "Tag_3" THEN
       "输出数据块".码垛升2 := TRUE;
       "输出数据块".平台升2 := TRUE;
       "输出数据块".回2 := TRUE;
       "输出数据块".码垛退2 := TRUE;
   END_IF;
END_REGION

REGION Network 2
   RUNG wire#powerrail
      Contact( "Tag_3" )
      wire#w1
      Contact( "输出数据块".码垛升2 )
      Contact( "码垛升到位传感器(h)" )
      R_Coil( "输出数据块".码垛升2 )
   END_RUNG
   RUNG wire#w1
      Contact( "输出数据块".平台升2 )
      Contact( "平台上到位传感器(0)" )
      R_Coil( "输出数据块".平台升2 )
   END_RUNG
   RUNG wire#w1
      Contact( "输出数据块".回2 )
      Contact( "回到位传感器(c)" )
      R_Coil( "输出数据块".回2 )
   END_RUNG
   RUNG wire#w1
      Contact( "输出数据块".码垛退2 )
      Contact( "退到位传感器(f)" )
      R_Coil( "输出数据块".码垛退2 )
   END_RUNG
   RUNG wire#powerrail
      Contact( "Tag_3" )
      I_Contact( "输出数据块".码垛升2 )
      I_Contact( "输出数据块".平台升2 )
      I_Contact( "输出数据块".回2 )
      I_Contact( "输出数据块".码垛退2 )
      Coil( "复位完成" )
   END_RUNG
   // the same network as SCL:
   IF "Tag_3" AND "输出数据块".码垛升2 AND "码垛升到位传感器(h)" THEN "输出数据块".码垛升2 := FALSE; END_IF;
   IF "Tag_3" AND "输出数据块".平台升2 AND "平台上到位传感器(0)" THEN "输出数据块".平台升2 := FALSE; END_IF;
   IF "Tag_3" AND "输出数据块".回2 AND "回到位传感器(c)" THEN "输出数据块".回2 := FALSE; END_IF;
   IF "Tag_3" AND "输出数据块".码垛退2 AND "退到位传感器(f)" THEN "输出数据块".码垛退2 := FALSE; END_IF;
   "复位完成" := "Tag_3" AND NOT "输出数据块".码垛升2 AND NOT "输出数据块".平台升2 AND NOT "输出数据块".回2 AND NOT "输出数据块".码垛退2;
END_REGION
END_FUNCTION

(* ===== HMI "HMI_RT_1" =====

HMI tags "默认变量表"
   "Tag_ScreenNumber" : UInt, internal

screen "画面_1" 800x480
   GraphicView "图形视图_1" at 0,0 size 801x480; Picture "屏幕截图 2024-04-17 131131"
*)